// ---- Interfaces/I_ManualTarget.TcIO
// Core §7.6.1 — a module that can be commanded by hand, reached by the SAME
// deterministic walk that already carries configuration writes (I_ConfigSource).
//
// This exists because the walk was missing and every Unit hand-wrote its own
// routing instead:
//
//     IF TargetPath = PressRam.Name THEN _M_RouteManual := PressRam.ManualCommand(...)
//     ELSIF TargetPath = Door.Name  THEN ...
//
// That is a call a project has to remember for correctness, which §1.1 O1 names
// as a framework defect rather than a project style. It failed exactly the way
// O1 predicts: the press registered eight children and routed three, so the
// feed axis, the two-hand control, the power group, the part sensor and the air
// monitor all published manual commands that the HMI rendered as buttons and
// the Unit refused, with no diagnostic anybody could act on. Nothing was wrong
// with those modules; the routing chain simply had no branch for them.
//
// Configuration never had this problem because it was built as a capability
// walk from the start: a module answers for its own Scope and the composite
// recurses. Manual commands now use the identical shape, so a registered child
// is commandable BECAUSE it is registered, and a new module type costs no
// routing code anywhere.
INTERFACE I_ManualTarget EXTENDS __System.IQueryInterface

// Apply one one-shot manual command to the module named by Scope. TRUE only
// from the module that owns the path AND accepted the value, so the walk
// continues past every module that is not the target. The owning module still
// validates the command against its own published catalogue (§5.6) — this
// carries the request, it does not privilege it.
METHOD M_ApplyManual : BOOL
VAR_INPUT
    Scope : STRING(255);
    Value : DINT;
END_VAR
END_METHOD

// §7.6.1a — apply one HELD manual request (hold-to-run) to the module named by
// Scope, carrying the enabling-device status the root derived from its §9
// safety facet.
//
// Enable travels WITH the request rather than being read by the module, because
// the fact belongs to the safety system and the root is where it is mirrored.
// A module that does not implement held commands inherits FB_ModuleBase's
// refusal, so an unsupported hold is a defined FALSE and never a silent no-op.
METHOD M_ApplyHeld : BOOL
VAR_INPUT
    Scope  : STRING(255);
    Value  : DINT;
    Enable : ST_ManualEnableStatus;
END_VAR
END_METHOD

END_INTERFACE

// ---- Interfaces/I_Module.TcIO
// Core §3.2 — everything a parent needs to discover, monitor, and roll up a child.
// Reconciliation vs. Core §3.2 text: no ErrorID property here (it would collide with
// the PLCopen ErrorID output every module exposes, Core §6.1); callers read
// GetFaultSummary().ReasonCode. GetFaultSummary returns ST_Diagnostic (Core §8.8),
// Recipe changeover is a prepare/commit/abort transaction (Core §3.8).
INTERFACE I_Module EXTENDS __System.IQueryInterface

METHOD Cyclic : BOOL
END_METHOD

// recursive first-out walk (Core §8.2, §6.9)
METHOD GetFaultSummary : ST_Diagnostic
END_METHOD

// Load/validate into staging only; active ParCfg remains unchanged.
METHOD PrepareRecipe : BOOL
VAR_INPUT
    Model : ST_ModelId;
END_VAR
END_METHOD

// Infallible bounded publication after a successful PrepareRecipe.
METHOD CommitRecipe
END_METHOD

METHOD AbortRecipe
END_METHOD

// Core §6.1/§8.3(b) — release a command the owner can no longer complete, so the
// inherited Execute-drop reset can clear a latched terminal state. A parent needs
// this generically: when a mode chain freezes on a fault it stops polling the
// children it commanded, and a child whose Execute stays asserted can never be
// re-issued (no rising edge) nor reset (the drop reset needs Execute low).
METHOD M_ReleaseCommand : BOOL
END_METHOD

PROPERTY FaultActive : BOOL
GET
END_GET
END_PROPERTY

// Core §6.1 — TRUE while the module is BUSY but deliberately not progressing
// because a declared condition is unsatisfied (ISA-88 HELD). It is NOT a fault:
// outputs are withdrawn, the reason is published at LOW severity, and progress
// resumes by itself when the condition returns. The parent reads this to explain
// the wait instead of reporting a generic stall (§6.9).
PROPERTY HoldActive : BOOL
GET
END_GET
END_PROPERTY

PROPERTY ModuleType : E_ModuleType
GET
END_GET
END_PROPERTY

PROPERTY Name : STRING(80)
GET
END_GET
END_PROPERTY

PROPERTY State : E_ExecState
GET
END_GET
END_PROPERTY

END_INTERFACE

// ---- Interfaces/I_Sequence.TcIO
// Core §6.8 — the sliver of a step chain its OWNER needs.
// A chain receives the host bridge at Setup (I_SequenceHost); this is the
// reverse direction, so FB_UnitBase can drive scan-scoped housekeeping for
// every attached chain without the project wiring a single call.
INTERFACE I_Sequence

// §6.10 one-scan reset of the shared transition result.
METHOD M_BeginScan
END_METHOD

// §6.8 the chain starts over at its first step, application state included
// (OnChainReset). Driven by the owning Unit at the transitions after which a
// chain can never resume: first scan, mode change, abort.
METHOD M_Restart
END_METHOD

// §6.9 the owning Unit left ERROR: re-arm the step that raised it so the
// chain re-evaluates the command state instead of resuming mid-handshake.
METHOD M_ResumeAfterError
END_METHOD

END_INTERFACE

// ---- Interfaces/I_SequenceHost.TcIO
// Core §6.7/§6.8 — the bridge from a separately-compiled sequence POU (SFC/ST/LD)
// to its owning module's protected framework services: step record, condition
// waits, run-style gate, part lifecycle, decisions, and completion/fault.
// FB_UnitBase implements it once; a sequence receives it at Setup. It carries
// framework plumbing ONLY — application decisions stay in the sequence's steps.
INTERFACE I_SequenceHost

// §6.11 publish a decision request
METHOD M_SequenceAskDecision
VAR_INPUT
    Req : ST_DecisionRequest;
END_VAR
END_METHOD

// §6.9(b) named plain-condition wait
METHOD M_SequenceAwait : BOOL
VAR_INPUT
    Idx : INT;
    Label : STRING(120);
    Ok : BOOL;
END_VAR
END_METHOD

// §6.11 withdraw an open request
METHOD M_SequenceClearDecision
END_METHOD

// §6.1 one-shot sequence completion (finite chains)
METHOD M_SequenceComplete
END_METHOD

// §8.11.2 carrier-less fallback counter
METHOD M_SequenceCountGood
END_METHOD

// §8.11.1 cycle-complete marker; FALSE = stop granted (chain must not loop)
METHOD M_SequenceEndOfCycle : BOOL
END_METHOD

// §6.9 first-out fault from a step
METHOD M_SequenceFault
VAR_INPUT
    Reason : E_Reason;
    DescriptionKey : STRING(255);
END_VAR
END_METHOD

// §3.16.3 EVENT_PART_PROCESSED (write-result-first; counts by verdict §8.11.2)
METHOD M_SequencePartProcessed : BOOL
VAR_INPUT
    Verdict : E_Verdict;
    Reason : E_Reason;
END_VAR
END_METHOD

// §3.16.3 EVENT_PART_RECEIVED
METHOD M_SequencePartReceived : BOOL
END_METHOD

// §3.16.1 measured value
METHOD M_SequencePartRecord : BOOL
VAR_INPUT
    RecordName : STRING(64);
    Value : LREAL;
    Minimum : LREAL;
    Maximum : LREAL;
    Target : LREAL;
    EngUnit : STRING(16);
END_VAR
END_METHOD

// §3.16.3 EVENT_PART_PROCESSING_STARTED
METHOD M_SequencePartStarted
END_METHOD

// §6.8 a chain announces itself at M_Attach so the owning Unit can run
// scan-scoped housekeeping for it. Idempotent: Setup may run more than once.
METHOD M_SequenceRegister : BOOL
VAR_INPUT
    Seq : I_Sequence;
END_VAR
END_METHOD

// §6.9 raise a first-out from a step, with the module path the §3.13 flow
// chart links to. Unlike M_SequenceFault this carries severity/category and a
// link, so a step can adopt a child's fault verbatim or declare its own message.
METHOD M_SequenceRaise : BOOL
VAR_INPUT
    Diag     : ST_Diagnostic;
    LinkPath : STRING(255);
END_VAR
END_METHOD

// §6.9(e) publish a message that informs and does NOT stop the chain: an
// AUTO_RESET come+gone event (§8.3(c)) plus the §3.13 flow-chart row mark.
METHOD M_SequenceWarn : BOOL
VAR_INPUT
    Diag : ST_Diagnostic;
END_VAR
END_METHOD

// §6.5 step record (feeds the §6.9 walk and the §8.11.4 profiler)
METHOD M_SequenceSetStep
VAR_INPUT
    StepNo : INT;
    StepName : STRING(120);
    Awaits : I_Module;
    AwaitingLabel : STRING(120);
    TimeClass : E_TimeClass;
    ExpectedTime : TIME;
    Branch : INT;                  // §6.12 concurrent leg, 0 = main line
END_VAR
END_METHOD

// §3.4.2 run-style pacing gate
METHOD M_SequenceStepGate : BOOL
VAR_INPUT
    Steppable : BOOL;
END_VAR
END_METHOD

// §3.4/§8.11 — accept a pending Stop BETWEEN cycles: abandon the open cycle
// profile (no §8.11.1 cycle is counted for a wait-only fragment) and complete.
METHOD M_SequenceStopNow
END_METHOD

// §3.4 — TRUE while a Stop is requested and the sequence still runs. A chain
// polls this at its between-cycles wait so a stop need not ride out a phantom cycle.
METHOD M_SequenceStopPending : BOOL
END_METHOD

// §6.11 consume the answer once (0 = none yet)
METHOD M_SequenceTakeDecision : INT
END_METHOD

END_INTERFACE

// ---- Interfaces/I_RecipeStore.TcIO
// Core §3.8a - a recipe provider whose records can be edited. Optional: a provider
// that implements it lets a root edit the recipe of ANY model it offers, not only
// the active one, and keeps an edit of the active model across a changeover.
// Found by __QUERYINTERFACE on the I_RecipeProvider a module was given.
INTERFACE I_RecipeStore

// Replace the record of exactly (ModelCode, RecipeKey) with Size bytes at pData.
// FALSE when that record does not exist or its size or SchemaVersion differs:
// a fallback record is never edited in a specific model's name.
METHOD Save : BOOL
VAR_INPUT
    ModelCode : STRING;
    RecipeKey : STRING;
    pData     : PVOID;
    Size      : UDINT;
END_VAR
END_METHOD

END_INTERFACE

// ---- Interfaces/I_RecipeProvider.TcIO
// Core §3.8 — pluggable recipe/type-data source. Implementations MUST validate
// completeness and SchemaVersion before filling ParCfg (migrate-or-fault; never partial).
// Queryable (like I_Module) so a root can ask a provider for I_RecipeStore (§3.8a).
INTERFACE I_RecipeProvider EXTENDS __System.IQueryInterface

// fills the caller's ParCfg; FALSE => caller faults with RECIPE_INVALID (Core §3.8)
METHOD Load : BOOL
VAR_INPUT
    ModelCode : STRING;
    RecipeKey : STRING;
    pParCfg : PVOID;
    Size    : UDINT;
END_VAR
END_METHOD

PROPERTY Ready : BOOL
GET
END_GET
END_PROPERTY

PROPERTY Source : E_RecipeSource
GET
END_GET
END_PROPERTY

END_INTERFACE

// ---- Connectivity/FB_LocalRecipeProvider.TcPOU
// Core §3.8 local provider. Validation is generic BECAUSE SchemaVersion is the
// first UINT of every ParCfg/record (§3.8): stored first-UINT must equal the
// target's initialized first-UINT, else Load = FALSE and the caller faults
// RECIPE_INVALID. Never a partial apply. Types stage through PrepareRecipe.
FUNCTION_BLOCK FB_LocalRecipeProvider IMPLEMENTS I_RecipeProvider, I_RecipeStore, I_RecipeCatalog
VAR PERSISTENT
    {attribute 'OPC.UA.DA' := '0'}
    _catalog : ST_LocalRecipeCatalog;
END_VAR
VAR
    _catalogInitialized : BOOL;
    _catalogRestoreVersion : UINT;
    _n    : INT;
    _models : ARRAY[1..PL_Fraktal.MAX_RECIPES] OF STRING(80);
    _keys   : ARRAY[1..PL_Fraktal.MAX_RECIPES] OF STRING(80);
    {attribute 'OPC.UA.DA' := '0'}
    _ptr  : ARRAY[1..PL_Fraktal.MAX_RECIPES] OF PVOID;
    _size : ARRAY[1..PL_Fraktal.MAX_RECIPES] OF UDINT;
END_VAR

// no cyclic body

METHOD Load : BOOL
VAR_INPUT
    ModelCode : STRING;
    RecipeKey : STRING;
    pParCfg : PVOID;
    Size    : UDINT;
END_VAR
VAR
    i, hit, fallback : INT;
    puT, puS : POINTER TO UINT;
END_VAR
_M_InitCatalog();
Load := FALSE;
IF (pParCfg = 0) OR (Size < SIZEOF(puT^)) THEN RETURN; END_IF
FOR i := 1 TO _catalog.Count DO
    IF (_catalog.Records[i].ModelCode = ModelCode)
    AND (_catalog.Records[i].RecipeKey = RecipeKey) THEN
        IF _catalog.Records[i].DataSize <> Size THEN RETURN; END_IF
        puT := pParCfg;
        puS := ADR(_catalog.Records[i].Data);
        IF puT^ <> puS^ THEN RETURN; END_IF
        MEMCPY(destAddr := pParCfg,
            srcAddr := ADR(_catalog.Records[i].Data), n := Size);
        Load := TRUE;
        RETURN;
    END_IF
END_FOR
hit := 0;
fallback := 0;
FOR i := 1 TO _n DO
    IF (_keys[i] = RecipeKey) AND (_models[i] = ModelCode) THEN
        hit := i;
        EXIT;
    ELSIF (_keys[i] = RecipeKey) AND (_models[i] = '') THEN
        fallback := i;
    END_IF
END_FOR
IF hit = 0 THEN
    hit := fallback;
END_IF
// Two statements, not one condition: IEC 61131-3 does not mandate short-circuit
// evaluation and TwinCAT's compile option for it is off by default, so a single
// `(hit = 0) OR (_size[hit] <> Size)` still reads _size[0] on the ordinary
// not-found path - out of bounds for ARRAY[1..MAX_RECIPES] (§3.8).
IF (hit = 0) OR (pParCfg = 0) THEN
    RETURN;                                       // unknown recipe -> caller faults (§3.8)
END_IF
IF _size[hit] <> Size THEN
    RETURN;                                       // size mismatch -> caller faults (§3.8)
END_IF
puT := pParCfg;
puS := _ptr[hit];
IF puT^ <> puS^ THEN
    RETURN;                                       // SchemaVersion mismatch: migrate-or-fault (§3.8)
END_IF
MEMCPY(destAddr := pParCfg, srcAddr := _ptr[hit], n := Size);
Load := TRUE;
END_METHOD

// I_RecipeStore - write an edited record back into the registered storage of
// exactly (ModelCode, RecipeKey). The fallback record is never edited in a
// specific model's name, and a size or SchemaVersion mismatch changes nothing.
METHOD Save : BOOL
VAR_INPUT
    ModelCode : STRING;
    RecipeKey : STRING;
    pData     : PVOID;
    Size      : UDINT;
END_VAR
VAR
    i, hit : INT;
    puT, puS : POINTER TO UINT;
END_VAR
_M_InitCatalog();
Save := FALSE;
IF (pData = 0) OR (Size < SIZEOF(puT^)) THEN RETURN; END_IF
FOR i := 1 TO _catalog.Count DO
    IF (_catalog.Records[i].ModelCode = ModelCode)
    AND (_catalog.Records[i].RecipeKey = RecipeKey) THEN
        IF _catalog.Records[i].DataSize <> Size THEN RETURN; END_IF
        puT := pData;
        puS := ADR(_catalog.Records[i].Data);
        IF puT^ <> puS^ THEN RETURN; END_IF
        MEMCPY(destAddr := ADR(_catalog.Records[i].Data),
            srcAddr := pData, n := Size);
        Save := TRUE;
        RETURN;
    END_IF
END_FOR
hit := 0;
FOR i := 1 TO _n DO
    IF (_keys[i] = RecipeKey) AND (_models[i] = ModelCode) THEN
        hit := i;
        EXIT;
    END_IF
END_FOR
IF (hit = 0) OR (pData = 0) THEN
    RETURN;
END_IF
IF _size[hit] <> Size THEN
    RETURN;
END_IF
puT := _ptr[hit];
puS := pData;
IF puT^ <> puS^ THEN
    RETURN;                                       // SchemaVersion differs: nothing written
END_IF
MEMCPY(destAddr := _ptr[hit], srcAddr := pData, n := Size);
Save := TRUE;
END_METHOD

// application wiring: one record per (ModelCode, RecipeKey); empty ModelCode is fallback.
METHOD Register : BOOL
VAR_INPUT
    ModelCode : STRING(80);
    RecipeKey : STRING(80);
    pData  : PVOID;
    Size   : UDINT;
END_VAR
VAR
    i : INT;
END_VAR
_M_InitCatalog();
IF (_n + _catalog.Count >= PL_Fraktal.MAX_RECIPES) OR (pData = 0) OR (RecipeKey = '') OR (Size < SIZEOF(UINT)) THEN
    Register := FALSE;
    RETURN;
END_IF
FOR i := 1 TO _n DO
    IF (_models[i] = ModelCode) AND (_keys[i] = RecipeKey) THEN
        Register := FALSE;
        RETURN;
    END_IF
END_FOR
FOR i := 1 TO _catalog.Count DO
    IF (_catalog.Records[i].ModelCode = ModelCode)
    AND (_catalog.Records[i].RecipeKey = RecipeKey) THEN
        Register := FALSE;
        RETURN;
    END_IF
END_FOR
_n := _n + 1;
_models[_n] := ModelCode;
_keys[_n]   := RecipeKey;
_ptr[_n]  := pData;
_size[_n] := Size;
Register := TRUE;
END_METHOD

PROPERTY Ready : BOOL
GET
Ready := (_n > 0);
END_GET
END_PROPERTY

PROPERTY Source : E_RecipeSource
GET
Source := E_RecipeSource.LOCAL;
END_GET
END_PROPERTY

METHOD PRIVATE _M_InitCatalog
VAR
    i, j : INT;
    schema : UINT;
    pSchema : POINTER TO UINT;
    valid : BOOL;
END_VAR
IF _catalogInitialized THEN RETURN; END_IF
_catalogInitialized := TRUE;
IF (_catalog.SchemaVersion = 1) AND (_catalog.Count >= 0)
AND (_catalog.Count <= PL_Fraktal.MAX_RECIPES) THEN
    valid := TRUE;
    FOR i := 1 TO _catalog.Count DO
        IF (_catalog.Records[i].SchemaVersion <> 1)
        OR (_catalog.Records[i].ModelCode = '') OR (_catalog.Records[i].RecipeKey = '')
        OR (_catalog.Records[i].DataSize < SIZEOF(schema))
        OR (_catalog.Records[i].DataSize > PL_Fraktal.MAX_MODEL_DATA_BYTES) THEN
            valid := FALSE;
        END_IF
        pSchema := ADR(_catalog.Records[i].Data);
        IF pSchema^ = 0 THEN valid := FALSE; END_IF
        FOR j := 1 TO i - 1 DO
            IF _catalog.Records[i].ModelCode = _catalog.Records[j].ModelCode THEN
                valid := FALSE;
            END_IF
        END_FOR
    END_FOR
    IF valid THEN RETURN; END_IF
END_IF
IF _catalog.SchemaVersion <> 0 THEN
    _catalogRestoreVersion := _catalog.SchemaVersion;
END_IF
_catalog.Count := 0;
_catalog.SchemaVersion := 1;
END_METHOD

METHOD M_ModelCount : INT
VAR_INPUT
    RecipeKey : STRING(80);
END_VAR
VAR
    i : INT;
END_VAR
_M_InitCatalog();
M_ModelCount := 0;
FOR i := 1 TO _n DO
    IF (_keys[i] = RecipeKey) AND (_models[i] <> '') THEN
        M_ModelCount := M_ModelCount + 1;
    END_IF
END_FOR
FOR i := 1 TO _catalog.Count DO
    IF _catalog.Records[i].RecipeKey = RecipeKey THEN
        M_ModelCount := M_ModelCount + 1;
    END_IF
END_FOR
END_METHOD

METHOD M_ModelCapacity : INT
VAR_INPUT
    RecipeKey : STRING(80);
END_VAR
VAR
    i : INT;
END_VAR
_M_InitCatalog();
M_ModelCapacity := M_ModelCount(RecipeKey := RecipeKey)
    + PL_Fraktal.MAX_RECIPES - _n - _catalog.Count;
// Released seed registration accepts 80 bytes; the root identity accepts 64.
// Preserve that API while refusing a catalog projection that would truncate it.
FOR i := 1 TO _n DO
    IF (_keys[i] = RecipeKey) AND (LEN(_models[i]) > 64) THEN
        M_ModelCapacity := 0; RETURN;
    END_IF
END_FOR
END_METHOD

METHOD M_ModelAt : BOOL
VAR_INPUT
    RecipeKey : STRING(80);
    Index : INT;
END_VAR
VAR_IN_OUT
    Id : ST_ModelId;
END_VAR
VAR
    i, ordinal : INT;
END_VAR
_M_InitCatalog();
M_ModelAt := FALSE;
IF Index < 1 THEN RETURN; END_IF
ordinal := 0;
FOR i := 1 TO _n DO
    IF (_keys[i] = RecipeKey) AND (_models[i] <> '') THEN
        ordinal := ordinal + 1;
        IF ordinal = Index THEN
            IF LEN(_models[i]) > 64 THEN RETURN; END_IF
            Id.ModelCode := _models[i];
            M_ModelAt := TRUE;
            RETURN;
        END_IF
    END_IF
END_FOR
FOR i := 1 TO _catalog.Count DO
    IF _catalog.Records[i].RecipeKey = RecipeKey THEN
        ordinal := ordinal + 1;
        IF ordinal = Index THEN
            Id.ModelCode := _catalog.Records[i].ModelCode;
            M_ModelAt := TRUE;
            RETURN;
        END_IF
    END_IF
END_FOR
END_METHOD

METHOD M_CreateModel : BOOL
VAR_INPUT
    ModelCode : STRING(64);
    RecipeKey : STRING(80);
    pData : PVOID;
    Size : UDINT;
END_VAR
VAR
    i, slot : INT;
    pSchema : POINTER TO UINT;
END_VAR
_M_InitCatalog();
M_CreateModel := FALSE;
IF (ModelCode = '') OR (RecipeKey = '') OR (pData = 0)
OR (Size < SIZEOF(pSchema^)) OR (Size > PL_Fraktal.MAX_MODEL_DATA_BYTES)
OR (_n + _catalog.Count >= PL_Fraktal.MAX_RECIPES) THEN RETURN; END_IF
pSchema := pData;
IF pSchema^ = 0 THEN RETURN; END_IF
FOR i := 1 TO _n DO
    IF _models[i] = ModelCode THEN RETURN; END_IF
END_FOR
FOR i := 1 TO _catalog.Count DO
    IF _catalog.Records[i].ModelCode = ModelCode THEN RETURN; END_IF
END_FOR
slot := _catalog.Count + 1;
_catalog.Records[slot].SchemaVersion := 1;
_catalog.Records[slot].ModelCode := ModelCode;
_catalog.Records[slot].RecipeKey := RecipeKey;
_catalog.Records[slot].DataSize := Size;
MEMCPY(destAddr := ADR(_catalog.Records[slot].Data), srcAddr := pData, n := Size);
_catalog.Count := slot; // publication LAST; every existing address stays stable
M_CreateModel := TRUE;
END_METHOD

METHOD M_TakeCatalogRestoreLoss : BOOL
VAR_OUTPUT
    Found : UINT;
END_VAR
_M_InitCatalog();
Found := _catalogRestoreVersion;
M_TakeCatalogRestoreLoss := Found <> 0;
_catalogRestoreVersion := 0;
END_METHOD

END_FUNCTION_BLOCK

// ---- Connectivity/FB_LocalAccessProvider.TcPOU
// Core §7.7(c) — DEFAULT local provider: a durable user table. Remote/central
// auth (server, LDAP via gateway) substitutes behind I_AccessProvider later.
//
// §14 - a PIN is never stored: each user keeps a random-per-registration salt and
// an iterated SHA-256 of salt and PIN, and the table is hidden from the ADS symbol
// table and OPC UA. Hiding is the control that matters for a short PIN - four
// digits fall to an offline search whatever the hash - so the hash's job is that a
// dump, backup or retained file does not hand the PINs out as text.
//
// TwinCAT restores PERSISTENT data by symbol and a hidden variable has none, so a
// hidden table cannot be PERSISTENT (IMPLEMENTATION_NOTES §154). The table is kept
// instead as one CRC-protected image document on an I_PersistMedium (§163): by
// default a file medium in the runtime's TwinCAT Boot directory, or the project's
// own medium (M_UseMedium) - which must be confidential, so a retentive-memory
// pool, readable over ADS, is refused. The medium keeps two copies, never
// overwrites the newest, and reports a document it confirmed and then lost. The
// owning root's FB_AccessManager drives restore and save through I_AccessStore
// every scan: a project calls nothing to make its users durable.
{attribute 'reflection'}
FUNCTION_BLOCK FB_LocalAccessProvider IMPLEMENTS I_AccessProvider, I_AccessStore
VAR_OUTPUT
    Restored     : BOOL;    // the retained table has been read (or there was none)
    Durable      : BOOL;    // every registration so far is in a written image
    StorageError : UDINT;   // last medium error (0 = none)
END_VAR
VAR
    {attribute 'hide'}
    {attribute 'OPC.UA.DA' := '0'}
    _users : ARRAY[1..PL_Fraktal.MAX_USERS] OF ST_UserRecord;
    {attribute 'hide'}
    {attribute 'OPC.UA.DA' := '0'}
    _n     : INT;
    {attribute 'hide'}
    _saltSeq : UDINT;
    // Transfer buffer: the image read, then each image written. It carries salts
    // and hashes, so it is hidden like the table; the medium only borrows it.
    {attribute 'hide'}
    {attribute 'OPC.UA.DA' := '0'}
    _image : ST_AccessImageV1;
    // '<project>.<path>.<instance>': hashed into the default key, so two providers -
    // or two PLC projects on one runtime - never share a document.
    {attribute 'instance-path'}
    {attribute 'noinit'}
    _instancePath : STRING(255);
    _key         : STRING(80);
    _keyChosen   : BOOL;            // the key is decided (possibly '' = volatile)
    {attribute 'OPC.UA.DA' := '0'}
    _medium      : I_PersistMedium; // injected, or _ownMedium
    {attribute 'OPC.UA.DA' := '0'}
    _ownMedium   : FB_FilePersistMedium;
    _ticket      : UDINT;
    _result      : ST_PersistResult;
    _phase       : INT;
    _generation  : UDINT;           // generation of the newest image written or read
    _restoreLost : BOOL;
    _dirty       : BOOL;            // the table changed since the last written image
    _changeSeq   : UDINT;
    _writeSeq    : UDINT;           // _changeSeq captured into the image being written
    _saveFailed  : BOOL;
    _readFailed  : BOOL;            // the medium could not answer the restore read
    _retry       : TON;
END_VAR
VAR CONSTANT
    IMAGE_MAGIC    : DWORD := DWORD#16#414B5246;   // 'FRKA', little endian
    RETRY_INTERVAL : TIME := T#10S;
END_VAR

// no cyclic body: the owning root's FB_AccessManager calls M_Service

// Keep the table on the project's medium instead of the Boot directory - the
// same instance the project gives its roots, so one line switches every
// retained document. Refused: no medium, a medium that is not confidential
// (a credential never becomes symbol-readable, §14), or a restore already begun.
METHOD M_UseMedium : BOOL
VAR_INPUT
    Medium : I_PersistMedium;
END_VAR
M_UseMedium := FALSE;
IF (_phase <> 0) OR (Medium = 0) THEN
    RETURN;
END_IF
IF NOT Medium.M_Confidential() THEN
    RETURN;
END_IF
_medium := Medium;
M_UseMedium := TRUE;
END_METHOD

// The table's document key on the medium (a file medium stores '<key>.a' and
// '<key>.b'). Without a call it is 'FraktalAccess_' and the CRC of this
// instance's path, so two providers - or two PLC projects on one runtime - never
// share a document. '' keeps the table volatile (a fixture, or a station whose
// users come from elsewhere). Letters, digits, '_', '.' and '-'. Refused once
// the restore has started: retargeting a live store would split one table.
METHOD M_UseKey : BOOL
VAR_INPUT
    Key : STRING(80);
END_VAR
M_UseKey := FALSE;
IF _phase <> 0 THEN
    RETURN;
END_IF
IF (Key <> '') AND NOT F_ValidPersistKey(Key := Key) THEN
    RETURN;
END_IF
_key := Key;
_keyChosen := TRUE;
M_UseKey := TRUE;
END_METHOD

// I_AccessStore - read the table's image once, then keep the written image
// current. A second root sharing this provider merely advances the same steps.
METHOD M_Service : BOOL
CASE _phase OF
    0:
        IF NOT _keyChosen THEN
            _key := _M_DefaultKey();
            _keyChosen := TRUE;
        END_IF
        IF _key = '' THEN
            Restored := TRUE;       // volatile by choice: nothing to restore or save
            Durable := FALSE;
            _phase := 90;
        ELSE
            IF _medium = 0 THEN
                _ownMedium.Setup(Folder := '', Where := Tc2_System.PATH_BOOTPATH);
                _medium := _ownMedium;
            END_IF
            _phase := 10;
        END_IF
    10:     // ask for the image
        MEMSET(destAddr := ADR(_image), fillByte := 0, n := SIZEOF(_image));
        _ticket := _medium.M_StartRead(Key := _key, pData := ADR(_image),
            Size := SIZEOF(_image));
        IF _ticket <> 0 THEN
            _phase := 11;
        END_IF
    11:
        IF _medium.M_Poll(Ticket := _ticket, Result := _result) THEN
            IF _result.Ok THEN
                _readFailed := FALSE;
                _M_FinishRestore();
                _phase := 30;
            ELSE
                // Not "no table": the medium could not answer. Asked again; until
                // then nothing is merged, written or claimed lost.
                _readFailed := TRUE;
                StorageError := _result.ErrorId;
                _retry(IN := FALSE, PT := RETRY_INTERVAL);
                _phase := 12;
            END_IF
        END_IF
    12:
        _retry(IN := TRUE, PT := RETRY_INTERVAL);
        IF _retry.Q THEN
            _retry(IN := FALSE, PT := RETRY_INTERVAL);
            _phase := 10;
        END_IF
    30:     // idle: rewrite the table whenever it changed
        _retry(IN := _saveFailed, PT := RETRY_INTERVAL);
        IF _dirty AND (NOT _saveFailed OR _retry.Q) THEN
            _retry(IN := FALSE, PT := RETRY_INTERVAL);
            _M_BuildImage();
            _phase := 40;
        END_IF
    40:
        _ticket := _medium.M_StartWrite(Key := _key, pData := ADR(_image),
            Size := SIZEOF(_image));
        IF _ticket <> 0 THEN
            _phase := 41;
        END_IF
    41:
        IF _medium.M_Poll(Ticket := _ticket, Result := _result) THEN
            _M_SaveDone(Ok := _result.Ok);
            _phase := 30;
        END_IF
    90:
        ;   // volatile: the table lives for this run only
ELSE
    _phase := 30;   // unknown step: idle again; a pending change is rewritten
END_CASE
M_Service := Restored;
END_METHOD

// Decide what the medium answered. A restore LOST something when the medium
// reports a document it confirmed and lost, when the image it returned does not
// validate, or when the image's users no longer fit. Nothing there and nothing
// confirmed is a first start. (A medium that could not answer is asked again.)
METHOD PRIVATE _M_FinishRestore
StorageError := _result.ErrorId;
_restoreLost := _result.Lost;
IF _result.Found THEN
    IF (_result.Length = SIZEOF(_image)) AND _M_ValidImage(Image := _image) THEN
        _generation := _image.Generation;
        IF NOT _M_Merge() THEN
            _restoreLost := TRUE;
        END_IF
    ELSE
        _restoreLost := TRUE;       // a document this build cannot read as a table
    END_IF
END_IF
MEMSET(destAddr := ADR(_image), fillByte := 0, n := SIZEOF(_image));
IF _restoreLost THEN
    // Write what survived as the new baseline: the loss is announced once, not at
    // every restart.
    _M_Changed();
END_IF
Restored := TRUE;
Durable := NOT _dirty;
END_METHOD

// A change made while the image was being written is newer than that image, so
// the table stays dirty and is written again.
METHOD PRIVATE _M_SaveDone
VAR_INPUT
    Ok : BOOL;
END_VAR
IF Ok THEN
    _generation := _image.Generation;
    _saveFailed := FALSE;
    StorageError := 0;
    IF _changeSeq = _writeSeq THEN
        _dirty := FALSE;
    END_IF
ELSE
    _saveFailed := TRUE;    // retried; the medium never overwrites the newest copy
    StorageError := _result.ErrorId;
END_IF
MEMSET(destAddr := ADR(_image), fillByte := 0, n := SIZEOF(_image));
Durable := NOT _dirty AND NOT _saveFailed;
END_METHOD

// 'FraktalAccess_' + the CRC-32 of this instance's path, in hexadecimal.
METHOD PRIVATE _M_DefaultKey : STRING(80)
VAR
    pathLength : UDINT;
END_VAR
pathLength := INT_TO_UDINT(LEN(_instancePath));
_M_DefaultKey := CONCAT('FraktalAccess_', Tc2_Utilities.DWORD_TO_HEXSTR(
    in := F_Crc32(pData := ADR(_instancePath), Size := pathLength),
    iPrecision := 8, bLoCase := FALSE));
END_METHOD

METHOD Authenticate : E_AccessLevel
VAR_INPUT
    User : STRING(32);
    Secret : STRING(32);
END_VAR
VAR
    i : INT;
    hit : INT;
    noSalt : ARRAY[0..15] OF BYTE;
    candidate : ARRAY[0..31] OF BYTE;
    diff : BYTE;
    k : INT;
END_VAR
Authenticate := E_AccessLevel.NONE;
hit := 0;
FOR i := 1 TO _n DO
    IF _users[i].User = User THEN
        hit := i;
    END_IF
END_FOR
IF hit = 0 THEN
    // An unknown user costs the same hash, so timing does not tell names apart.
    _M_Hash(Salt := noSalt, Pin := Secret, Digest := candidate);
    RETURN;
END_IF
_M_Hash(Salt := _users[hit].Salt, Pin := Secret, Digest := candidate);
diff := 0;
FOR k := 0 TO 31 DO
    diff := diff OR (candidate[k] XOR _users[hit].PinHash[k]);
END_FOR
IF diff = 0 THEN
    Authenticate := _users[hit].Level;
END_IF
END_METHOD

// commissioning-time user entry (itself an ACCESS_POLICY-gated edit via the HMI).
// Idempotent by User: re-registering replaces PIN/level, and the retained table
// keeps the user, so a composition root may register its defaults every boot
// without duplicates. Every registration draws a new salt. A registration made
// before the restore completes is kept and wins over the retained record.
// Refused: an empty name, a level outside NONE..ADMIN, or a full table.
METHOD Register : BOOL
VAR_INPUT
    User : STRING(32);
    Pin : STRING(32);
    Level : E_AccessLevel;
END_VAR
VAR
    i : INT;
    slot : INT;
END_VAR
Register := FALSE;
IF (User = '') OR (TO_DINT(Level) < TO_DINT(E_AccessLevel.NONE))
OR (TO_DINT(Level) > TO_DINT(E_AccessLevel.ADMIN)) THEN
    RETURN;     // an image holding such a record would be refused at restore
END_IF
slot := 0;
FOR i := 1 TO _n DO
    IF _users[i].User = User THEN
        slot := i;
    END_IF
END_FOR
IF slot = 0 THEN
    IF _n >= PL_Fraktal.MAX_USERS THEN
        RETURN;
    END_IF
    _n := _n + 1;
    slot := _n;
    _users[slot].User := User;
END_IF
_M_NewSalt(User := User, Salt := _users[slot].Salt);
_M_Hash(Salt := _users[slot].Salt, Pin := Pin, Digest := _users[slot].PinHash);
_users[slot].Level := Level;
_M_Changed();
Register := TRUE;
END_METHOD

METHOD M_RestoreLost : BOOL
M_RestoreLost := _restoreLost;
END_METHOD

METHOD M_SaveFailed : BOOL
M_SaveFailed := _saveFailed OR _readFailed;
END_METHOD

// Add every retained user not registered in this run. A registration made before
// the restore finished is newer, so it stands. FALSE = a user did not fit.
METHOD PRIVATE _M_Merge : BOOL
VAR
    i : INT;
    k : INT;
    found : BOOL;
END_VAR
_M_Merge := TRUE;
FOR i := 1 TO _image.Count DO
    found := FALSE;
    FOR k := 1 TO _n DO
        IF _users[k].User = _image.Users[i].User THEN
            found := TRUE;
        END_IF
    END_FOR
    IF NOT found THEN
        IF _n < PL_Fraktal.MAX_USERS THEN
            _n := _n + 1;
            _users[_n] := _image.Users[i];
        ELSE
            _M_Merge := FALSE;
        END_IF
    END_IF
END_FOR
END_METHOD

// Whole-image validation: format, checksum, then every record. One bad record
// rejects the image - a table is restored completely or not at all.
METHOD PRIVATE _M_ValidImage : BOOL
VAR_IN_OUT
    Image : ST_AccessImageV1;
END_VAR
VAR
    i : INT;
    k : INT;
END_VAR
_M_ValidImage := FALSE;
IF (Image.SchemaVersion <> 1) OR (Image.ByteCount <> SIZEOF(Image))
OR (Image.Magic <> IMAGE_MAGIC) OR (Image.Reserved <> 0)
OR (Image.Count < 0) OR (Image.Count > PL_Fraktal.MAX_USERS) THEN
    RETURN;
END_IF
IF Image.Crc <> F_Crc32(pData := ADR(Image), Size := SIZEOF(Image) - SIZEOF(Image.Crc)) THEN
    RETURN;
END_IF
FOR i := 1 TO Image.Count DO
    IF (Image.Users[i].User = '')
    OR (TO_DINT(Image.Users[i].Level) < TO_DINT(E_AccessLevel.NONE))
    OR (TO_DINT(Image.Users[i].Level) > TO_DINT(E_AccessLevel.ADMIN)) THEN
        RETURN;
    END_IF
    FOR k := 1 TO i - 1 DO
        IF Image.Users[k].User = Image.Users[i].User THEN
            RETURN;
        END_IF
    END_FOR
END_FOR
_M_ValidImage := TRUE;
END_METHOD

METHOD PRIVATE _M_BuildImage
VAR
    i : INT;
END_VAR
MEMSET(destAddr := ADR(_image), fillByte := 0, n := SIZEOF(_image));
_image.SchemaVersion := 1;
_image.ByteCount := TO_UINT(SIZEOF(_image));
_image.Magic := IMAGE_MAGIC;
_image.Generation := _generation + 1;
_image.Count := _n;
FOR i := 1 TO _n DO
    _image.Users[i] := _users[i];
END_FOR
_image.Crc := F_Crc32(pData := ADR(_image), Size := SIZEOF(_image) - SIZEOF(_image.Crc));
_writeSeq := _changeSeq;
END_METHOD

METHOD PRIVATE _M_Changed
_dirty := TRUE;
_changeSeq := _changeSeq + 1;
Durable := FALSE;
END_METHOD

// A salt unique to this registration: the clock, a sequence and the user name,
// hashed. It need not be secret, only never repeated.
METHOD PRIVATE _M_NewSalt
VAR_INPUT
    User : STRING(32);
END_VAR
VAR_IN_OUT
    Salt : ARRAY[0..15] OF BYTE;
END_VAR
VAR
    seed : ARRAY[0..47] OF BYTE;
    now : ULINT;
    digest : ARRAY[0..31] OF BYTE;
END_VAR
now := Tc2_Utilities.F_GetSystemTime();
_saltSeq := _saltSeq + 1;
MEMCPY(destAddr := ADR(seed), srcAddr := ADR(now), n := SIZEOF(now));
MEMCPY(destAddr := ADR(seed) + 8, srcAddr := ADR(_saltSeq), n := SIZEOF(_saltSeq));
MEMCPY(destAddr := ADR(seed) + 12, srcAddr := ADR(User), n := INT_TO_UDINT(LEN(User)));
F_Sha256(pData := ADR(seed), Size := 12 + INT_TO_UDINT(LEN(User)), Digest := digest);
MEMCPY(destAddr := ADR(Salt), srcAddr := ADR(digest), n := 16);
END_METHOD

// SHA-256(Salt || Pin), then PL_Fraktal.PIN_HASH_ROUNDS more rounds of
// SHA-256(previous || Salt).
METHOD PRIVATE _M_Hash
VAR_INPUT
    Pin : STRING(32);
END_VAR
VAR_IN_OUT
    Salt   : ARRAY[0..15] OF BYTE;
    Digest : ARRAY[0..31] OF BYTE;
END_VAR
VAR
    buf : ARRAY[0..47] OF BYTE;
    round : UINT;
END_VAR
MEMCPY(destAddr := ADR(buf), srcAddr := ADR(Salt), n := 16);
MEMCPY(destAddr := ADR(buf) + 16, srcAddr := ADR(Pin), n := INT_TO_UDINT(LEN(Pin)));
F_Sha256(pData := ADR(buf), Size := 16 + INT_TO_UDINT(LEN(Pin)), Digest := Digest);
FOR round := 1 TO PL_Fraktal.PIN_HASH_ROUNDS DO
    MEMCPY(destAddr := ADR(buf), srcAddr := ADR(Digest), n := 32);
    MEMCPY(destAddr := ADR(buf) + 32, srcAddr := ADR(Salt), n := 16);
    F_Sha256(pData := ADR(buf), Size := 48, Digest := Digest);
END_FOR
MEMSET(destAddr := ADR(buf), fillByte := 0, n := SIZEOF(buf));
END_METHOD

END_FUNCTION_BLOCK

// ---- Platform/FB_FilePersistMedium.TcPOU
// Core §3.8b - the FILE medium (E_ConfigStore.FILE_JSON) on Tc2_System file
// services. Each key is two files in one folder, '<key>.a' and '<key>.b', and a
// write always replaces the slot NOT holding the newest valid copy, so a write
// cut short by a power loss leaves the previous document whole.
//
// Every file is an 80-byte text header line, then the document unchanged:
//   FRAKTAL-DOC 1 G=<generation> L=<length> K=<key CRC> C=<data CRC> H=<header CRC>
// in hexadecimal, so a set document stays readable in an editor. K binds a file
// to its key (a copy renamed to another key is refused), C checks the document
// and H the header. The highest valid generation wins on read.
//
// Both headers are read again before every write: the slot to replace and the
// next generation always come from what is on storage NOW, never from an earlier
// conclusion. A slot that cannot be READ (a file-service error other than "not
// found") is not a slot that is empty: a read then answers Ok = FALSE - the
// medium could not answer, nothing is claimed lost - and a write is refused
// without touching either file. Only content that reads but does not verify is
// treated as damaged.
//
// The generation each key was last CONFIRMED written at is kept PERSISTENT
// (it is not secret). A read that finds nothing valid where something was
// confirmed, or finds an older generation, reports Lost. TwinCAT stores the
// table at shutdown or on an explicit persistent write, so it can lag and never
// vouches for a write that did not happen; a stale marker can only miss a loss.
// The table is keyed by F_Crc32(folder + key), so retargeting the medium never
// claims a loss for files that were simply never written there. Keys beyond
// MAX_PERSIST_KEYS still work, without loss detection.
//
// Not symbol-readable: documents pass through the caller's buffer, so this
// medium may hold credentials (M_Confidential). On an IPC image with a write
// filter (UWF/EWF/FBWF), the folder must be excluded or every write reverts at
// the next boot. Files are created by the TwinCAT runtime's account; the
// folder's ACL decides who else may change them.
FUNCTION_BLOCK FB_FilePersistMedium EXTENDS FB_PersistMediumBase
VAR_OUTPUT
    StorageError : UDINT;   // last file-service error (0 = none)
END_VAR
VAR PERSISTENT
    {attribute 'OPC.UA.DA' := '0'}
    _confirmedKey : ARRAY[1..PL_Fraktal.MAX_PERSIST_KEYS] OF DWORD;
    {attribute 'OPC.UA.DA' := '0'}
    _confirmedGen : ARRAY[1..PL_Fraktal.MAX_PERSIST_KEYS] OF UDINT;
END_VAR
VAR
    _folder      : STRING(160);
    _where       : Tc2_System.E_OpenPath := Tc2_System.PATH_BOOTPATH;
    _foldersMade : BOOL;
    _mkPos       : INT;
    // The active request.
    _phase    : INT;
    _keyCrc   : DWORD;
    _slot     : INT;
    _hdrValid : ARRAY[1..2] OF BOOL;
    _hdrGen   : ARRAY[1..2] OF UDINT;
    _hdrLen   : ARRAY[1..2] OF UDINT;
    _hdrCrc   : ARRAY[1..2] OF DWORD;
    _invalidSeen : BOOL;    // a slot read but did not verify
    _ioFailed : BOOL;       // a slot could not be read at all
    _attempt  : INT;
    _ioOk     : BOOL;
    _handle   : UINT;
    _newGen   : UDINT;
    _header   : ARRAY[0..79] OF BYTE;   // read into / written from
    _expect   : ARRAY[0..79] OF BYTE;   // the header a read one must equal
    {attribute 'OPC.UA.DA' := '0'}
    _mkdir : Tc2_System.FB_CreateDir;
    {attribute 'OPC.UA.DA' := '0'}
    _open  : Tc2_System.FB_FileOpen;
    {attribute 'OPC.UA.DA' := '0'}
    _read  : Tc2_System.FB_FileRead;
    {attribute 'OPC.UA.DA' := '0'}
    _write : Tc2_System.FB_FileWrite;
    {attribute 'OPC.UA.DA' := '0'}
    _close : Tc2_System.FB_FileClose;
END_VAR
VAR CONSTANT
    HEADER_BYTES   : UDINT := 80;
    HEADER_TEXT    : STRING(80) := 'FRAKTAL-DOC 1 G=00000000 L=00000000 K=00000000 C=00000000 H=00000000';
    HEADER_CRC_SPAN : UDINT := 58;      // bytes before 'H='
    FILE_NOT_FOUND : UDINT := 16#70C;   // ADSERR_DEVICE_NOTFOUND
    CLOSE_DONE     : UDINT := 16#703;   // the handle is already released
    TOO_LARGE      : UDINT := 16#705;   // the document exceeds the caller's buffer
    IO_TIMEOUT     : TIME := T#3S;
END_VAR

// no cyclic body: every caller's M_Poll advances the medium

// Where the files live. Where = PATH_GENERIC takes an absolute Folder, for
// example 'C:\ProgramData\Fraktal\Station\'; PATH_BOOTPATH is relative to the
// TwinCAT Boot directory ('' = the directory itself). Missing folders are
// created on the first request. At most 160 characters; a trailing separator is
// added. Refused once a request was queued: one medium never splits a document
// over two folders.
METHOD Setup : BOOL
VAR_INPUT
    Folder : STRING(200);
    Where  : Tc2_System.E_OpenPath;
END_VAR
VAR
    n : INT;
    p : POINTER TO BYTE;
END_VAR
Setup := FALSE;
IF (_lastTicket > 0) OR (LEN(Folder) > 159) THEN
    RETURN;
END_IF
_folder := Folder;
n := LEN(_folder);
IF n > 0 THEN
    p := ADR(_folder);
    IF (p[n - 1] <> 92) AND (p[n - 1] <> 47) THEN
        _folder := CONCAT(_folder, '\');
    END_IF
END_IF
_where := Where;
_foldersMade := FALSE;
_mkPos := 0;
Setup := TRUE;
END_METHOD

METHOD M_Kind : E_ConfigStore
M_Kind := E_ConfigStore.FILE_JSON;
END_METHOD

METHOD M_Confidential : BOOL
M_Confidential := TRUE;
END_METHOD

METHOD PROTECTED _M_Step : BOOL
VAR
    i : INT;
    best : INT;
    confirmed : UDINT;
    keyPath : STRING(255);
END_VAR
_M_Step := FALSE;
CASE _phase OF
    0:      // a new request: read both headers first, for a read and a write alike
        IF NOT _foldersMade THEN
            _phase := 1;
            RETURN;
        END_IF
        keyPath := CONCAT(_folder, _qKey[_active]);
        _keyCrc := F_Crc32(pData := ADR(keyPath), Size := INT_TO_UDINT(LEN(keyPath)));
        _invalidSeen := FALSE;
        _ioFailed := FALSE;
        FOR i := 1 TO 2 DO
            _hdrValid[i] := FALSE;
        END_FOR
        _slot := 1;
        _phase := 10;
    1:      // create the folder chain, one level per operation
        i := _M_NextSeparator(StartAt := _mkPos);
        IF i < 0 THEN
            _foldersMade := TRUE;
            _phase := 0;
        ELSE
            _mkPos := i + 1;
            _mkdir(bExecute := FALSE);
            _mkdir(sNetId := '', sPathName := LEFT(_folder, i), ePath := _where,
                bExecute := TRUE, tTimeout := IO_TIMEOUT);
            _phase := 2;
        END_IF
    2:
        _mkdir(bExecute := FALSE);
        IF NOT _mkdir.bBusy THEN
            _phase := 1;            // an existing folder answers with an error: ignored
        END_IF

    10:     // header scan: open the slot
        _open(bExecute := FALSE);
        _open(sNetId := '', sPathName := _M_Path(Slot := _slot),
            nMode := Tc2_System.FOPEN_MODEREAD OR Tc2_System.FOPEN_MODEBINARY,
            ePath := _where, bExecute := TRUE, tTimeout := IO_TIMEOUT);
        _phase := 11;
    11:
        _open(bExecute := FALSE);
        IF NOT _open.bBusy THEN
            IF _open.bError THEN
                IF _open.nErrId <> FILE_NOT_FOUND THEN
                    _M_IoFailed(ErrorId := _open.nErrId);   // there, but not readable
                END_IF
                _phase := 16;
            ELSE
                _handle := _open.hFile;
                _phase := 12;
            END_IF
        END_IF
    12:
        MEMSET(destAddr := ADR(_header), fillByte := 0, n := HEADER_BYTES);
        _read(bExecute := FALSE);
        _read(sNetId := '', hFile := _handle, pReadBuff := ADR(_header),
            cbReadLen := HEADER_BYTES, bExecute := TRUE, tTimeout := IO_TIMEOUT);
        _phase := 13;
    13:
        _read(bExecute := FALSE);
        IF NOT _read.bBusy THEN
            IF _read.bError THEN
                _M_IoFailed(ErrorId := _read.nErrId);
            ELSE
                // A short file or a header that does not verify is damaged content.
                _hdrValid[_slot] := (_read.cbRead = HEADER_BYTES) AND _M_ParseHeader(Slot := _slot);
                IF NOT _hdrValid[_slot] THEN
                    _invalidSeen := TRUE;
                END_IF
            END_IF
            _phase := 14;
        END_IF
    14:
        _close(bExecute := FALSE);
        _close(sNetId := '', hFile := _handle, bExecute := TRUE, tTimeout := IO_TIMEOUT);
        _phase := 15;
    15:
        _close(bExecute := FALSE);
        IF NOT _close.bBusy THEN
            IF _close.bError AND (_close.nErrId <> CLOSE_DONE) THEN
                StorageError := _close.nErrId;
                _phase := 14;                       // never leak an open handle
            ELSE
                _handle := 0;
                _phase := 16;
            END_IF
        END_IF
    16:
        IF _slot = 1 THEN
            _slot := 2;
            _phase := 10;
        ELSIF _ioFailed THEN
            // Storage did not answer: never conclude "empty" from that, and never
            // write over a copy that could not be read.
            _qResult[_active].ErrorId := StorageError;
            _M_Finish();
            _M_Step := TRUE;
        ELSIF _qWrite[_active] THEN
            _phase := 40;
        ELSE
            _attempt := 0;
            _phase := 30;
        END_IF

    30:     // read the newest slot still valid; a rejected slot is no longer valid
        IF _attempt < 2 THEN
            _slot := _M_Newest();
        ELSE
            _slot := 0;
        END_IF
        confirmed := _M_ConfirmedGen();
        IF _slot = 0 THEN
            // Nothing valid. Lost when something existed or was confirmed.
            _qResult[_active].Ok := TRUE;
            _qResult[_active].Lost := _invalidSeen OR (confirmed > 0);
            _M_Finish();
            _M_Step := TRUE;
        ELSIF _hdrLen[_slot] > _qSize[_active] THEN
            _qResult[_active].ErrorId := TOO_LARGE;
            _M_Finish();
            _M_Step := TRUE;
        ELSIF _hdrLen[_slot] = 0 THEN
            // A deletion record: nothing there, by intent.
            _qResult[_active].Ok := TRUE;
            _qResult[_active].Lost := confirmed > _hdrGen[_slot];
            _M_Finish();
            _M_Step := TRUE;
        ELSE
            _phase := 31;
        END_IF
    31:
        _open(bExecute := FALSE);
        _open(sNetId := '', sPathName := _M_Path(Slot := _slot),
            nMode := Tc2_System.FOPEN_MODEREAD OR Tc2_System.FOPEN_MODEBINARY,
            ePath := _where, bExecute := TRUE, tTimeout := IO_TIMEOUT);
        _phase := 32;
    32:
        _open(bExecute := FALSE);
        IF NOT _open.bBusy THEN
            IF _open.bError THEN
                _M_IoFailed(ErrorId := _open.nErrId);
                _qResult[_active].ErrorId := StorageError;
                _M_Finish();
                _M_Step := TRUE;
            ELSE
                _handle := _open.hFile;
                _phase := 33;
            END_IF
        END_IF
    33:
        _read(bExecute := FALSE);
        _read(sNetId := '', hFile := _handle, pReadBuff := ADR(_header),
            cbReadLen := HEADER_BYTES, bExecute := TRUE, tTimeout := IO_TIMEOUT);
        _phase := 34;
    34:
        _read(bExecute := FALSE);
        IF NOT _read.bBusy THEN
            IF _read.bError THEN
                _M_IoFailed(ErrorId := _read.nErrId);
                _ioOk := FALSE;
                _phase := 37;
            ELSE
                // The header must still be the one the scan accepted for THIS slot.
                _M_BuildHeader(pDst := ADR(_expect), Generation := _hdrGen[_slot],
                    Length := _hdrLen[_slot], DataCrc := _hdrCrc[_slot]);
                _ioOk := (_read.cbRead = HEADER_BYTES)
                    AND (MEMCMP(pBuf1 := ADR(_header), pBuf2 := ADR(_expect), n := HEADER_BYTES) = 0);
                IF _ioOk THEN
                    _phase := 35;
                ELSE
                    _phase := 37;
                END_IF
            END_IF
        END_IF
    35:
        _read(bExecute := FALSE);
        _read(sNetId := '', hFile := _handle, pReadBuff := _qData[_active],
            cbReadLen := _hdrLen[_slot], bExecute := TRUE, tTimeout := IO_TIMEOUT);
        _phase := 36;
    36:
        _read(bExecute := FALSE);
        IF NOT _read.bBusy THEN
            IF _read.bError THEN
                _M_IoFailed(ErrorId := _read.nErrId);
                _ioOk := FALSE;
            ELSE
                _ioOk := (_read.cbRead = _hdrLen[_slot]);
            END_IF
            _phase := 37;
        END_IF
    37:
        _close(bExecute := FALSE);
        _close(sNetId := '', hFile := _handle, bExecute := TRUE, tTimeout := IO_TIMEOUT);
        _phase := 38;
    38:
        _close(bExecute := FALSE);
        IF NOT _close.bBusy THEN
            IF _close.bError AND (_close.nErrId <> CLOSE_DONE) THEN
                StorageError := _close.nErrId;
                _phase := 37;
            ELSE
                _handle := 0;
                IF _ioFailed THEN
                    _qResult[_active].ErrorId := StorageError;
                    _M_Finish();
                    _M_Step := TRUE;
                ELSIF _ioOk AND (F_Crc32(pData := _qData[_active], Size := _hdrLen[_slot])
                        = _hdrCrc[_slot]) THEN
                    _qResult[_active].Ok := TRUE;
                    _qResult[_active].Found := TRUE;
                    _qResult[_active].Length := _hdrLen[_slot];
                    _qResult[_active].Lost := _M_ConfirmedGen() > _hdrGen[_slot];
                    StorageError := 0;
                    _M_Finish();
                    _M_Step := TRUE;
                ELSE
                    _M_RejectSlot();            // damaged content: try the other slot
                END_IF
            END_IF
        END_IF

    40:     // write into the slot not holding the newest valid copy
        best := _M_Newest();
        _slot := 1;
        IF best = 1 THEN
            _slot := 2;
        END_IF
        _newGen := _M_ConfirmedGen();
        FOR i := 1 TO 2 DO
            IF _hdrValid[i] THEN
                _newGen := MAX(_newGen, _hdrGen[i]);
            END_IF
        END_FOR
        _newGen := _newGen + 1;
        _M_BuildHeader(pDst := ADR(_header), Generation := _newGen, Length := _qSize[_active],
            DataCrc := F_Crc32(pData := _qData[_active], Size := _qSize[_active]));
        _ioOk := TRUE;
        _phase := 41;
    41:
        _open(bExecute := FALSE);
        _open(sNetId := '', sPathName := _M_Path(Slot := _slot),
            nMode := Tc2_System.FOPEN_MODEWRITE OR Tc2_System.FOPEN_MODEBINARY,
            ePath := _where, bExecute := TRUE, tTimeout := IO_TIMEOUT);
        _phase := 42;
    42:
        _open(bExecute := FALSE);
        IF NOT _open.bBusy THEN
            IF _open.bError THEN
                StorageError := _open.nErrId;
                _qResult[_active].ErrorId := _open.nErrId;
                _M_Finish();
                _M_Step := TRUE;
            ELSE
                _handle := _open.hFile;
                _phase := 43;
            END_IF
        END_IF
    43:
        _write(bExecute := FALSE);
        _write(sNetId := '', hFile := _handle, pWriteBuff := ADR(_header),
            cbWriteLen := HEADER_BYTES, bExecute := TRUE, tTimeout := IO_TIMEOUT);
        _phase := 44;
    44:
        _write(bExecute := FALSE);
        IF NOT _write.bBusy THEN
            _ioOk := NOT _write.bError AND (_write.cbWrite = HEADER_BYTES);
            IF _write.bError THEN
                StorageError := _write.nErrId;
            END_IF
            IF _ioOk AND (_qSize[_active] > 0) THEN
                _phase := 45;
            ELSE
                _phase := 47;
            END_IF
        END_IF
    45:
        _write(bExecute := FALSE);
        _write(sNetId := '', hFile := _handle, pWriteBuff := _qData[_active],
            cbWriteLen := _qSize[_active], bExecute := TRUE, tTimeout := IO_TIMEOUT);
        _phase := 46;
    46:
        _write(bExecute := FALSE);
        IF NOT _write.bBusy THEN
            _ioOk := NOT _write.bError AND (_write.cbWrite = _qSize[_active]);
            IF _write.bError THEN
                StorageError := _write.nErrId;
            END_IF
            _phase := 47;
        END_IF
    47:
        _close(bExecute := FALSE);
        _close(sNetId := '', hFile := _handle, bExecute := TRUE, tTimeout := IO_TIMEOUT);
        _phase := 48;
    48:
        _close(bExecute := FALSE);
        IF NOT _close.bBusy THEN
            IF _close.bError AND (_close.nErrId <> CLOSE_DONE) THEN
                StorageError := _close.nErrId;
                _phase := 47;
            ELSE
                _handle := 0;
                // Durable only if the handle closed cleanly as well.
                IF _ioOk AND NOT _close.bError THEN
                    _M_Confirm();
                    _qResult[_active].Ok := TRUE;
                    StorageError := 0;
                ELSE
                    _qResult[_active].ErrorId := StorageError;
                END_IF
                _M_Finish();
                _M_Step := TRUE;
            END_IF
        END_IF
ELSE
    _qResult[_active].ErrorId := INVALID_REQUEST;   // unknown step: fail the request
    _M_Finish();
    _M_Step := TRUE;
END_CASE
END_METHOD

METHOD PRIVATE _M_Finish
IF NOT _qResult[_active].Ok AND (_qResult[_active].ErrorId = 0) THEN
    _qResult[_active].ErrorId := INVALID_REQUEST;
END_IF
_phase := 0;
END_METHOD

// A slot could not be read at all: the request cannot conclude anything about it.
METHOD PRIVATE _M_IoFailed
VAR_INPUT
    ErrorId : UDINT;
END_VAR
_ioFailed := TRUE;
StorageError := ErrorId;
END_METHOD

// The slot's document did not verify: it is damaged, so it stops being a
// candidate and the newest remaining valid slot is tried.
METHOD PRIVATE _M_RejectSlot
_invalidSeen := TRUE;
_hdrValid[_slot] := FALSE;
_attempt := _attempt + 1;
_phase := 30;
END_METHOD

// The slot with the highest valid header generation, 0 when neither is valid.
METHOD PRIVATE _M_Newest : INT
_M_Newest := 0;
IF _hdrValid[1] THEN
    _M_Newest := 1;
END_IF
IF _hdrValid[2] THEN
    IF _M_Newest = 0 THEN
        _M_Newest := 2;
    ELSIF _hdrGen[2] > _hdrGen[1] THEN
        _M_Newest := 2;
    END_IF
END_IF
END_METHOD

// Record the generation just written for this key (the persistent marker).
METHOD PRIVATE _M_Confirm
VAR
    i : INT;
END_VAR
FOR i := 1 TO PL_Fraktal.MAX_PERSIST_KEYS DO
    IF (_confirmedGen[i] > 0) AND (_confirmedKey[i] = _keyCrc) THEN
        _confirmedGen[i] := _newGen;
        RETURN;
    END_IF
END_FOR
FOR i := 1 TO PL_Fraktal.MAX_PERSIST_KEYS DO
    IF _confirmedGen[i] = 0 THEN
        _confirmedKey[i] := _keyCrc;
        _confirmedGen[i] := _newGen;
        RETURN;
    END_IF
END_FOR
END_METHOD

METHOD PRIVATE _M_ConfirmedGen : UDINT
VAR
    i : INT;
END_VAR
_M_ConfirmedGen := 0;
FOR i := 1 TO PL_Fraktal.MAX_PERSIST_KEYS DO
    IF (_confirmedGen[i] > 0) AND (_confirmedKey[i] = _keyCrc) THEN
        _M_ConfirmedGen := _confirmedGen[i];
        RETURN;
    END_IF
END_FOR
END_METHOD

METHOD PRIVATE _M_Path : STRING(255)
VAR_INPUT
    Slot : INT;
END_VAR
IF Slot = 2 THEN
    _M_Path := CONCAT(CONCAT(_folder, _qKey[_active]), '.b');
ELSE
    _M_Path := CONCAT(CONCAT(_folder, _qKey[_active]), '.a');
END_IF
END_METHOD

// Position of the next '\' or '/' at or after StartAt that ends a folder to create,
// -1 when none is left. A drive root ('C:\') and a leading UNC prefix are skipped.
METHOD PRIVATE _M_NextSeparator : INT
VAR_INPUT
    StartAt : INT;
END_VAR
VAR
    p : POINTER TO BYTE;
    i : INT;
END_VAR
_M_NextSeparator := -1;
p := ADR(_folder);
FOR i := MAX(StartAt, 0) TO 159 DO
    IF p[i] = 0 THEN
        RETURN;
    END_IF
    IF ((p[i] = 92) OR (p[i] = 47)) AND (i > 2) THEN
        _M_NextSeparator := i;
        RETURN;
    END_IF
END_FOR
END_METHOD

METHOD PRIVATE _M_BuildHeader
VAR_INPUT
    pDst       : POINTER TO BYTE;
    Generation : UDINT;
    Length     : UDINT;
    DataCrc    : DWORD;
END_VAR
VAR
    text : STRING(80);
END_VAR
text := HEADER_TEXT;
MEMSET(destAddr := pDst, fillByte := 32, n := HEADER_BYTES);
MEMCPY(destAddr := pDst, srcAddr := ADR(text), n := INT_TO_UDINT(LEN(text)));
pDst[HEADER_BYTES - 1] := 10;
_M_PutHex(pDst := pDst + 16, Value := UDINT_TO_DWORD(Generation));
_M_PutHex(pDst := pDst + 27, Value := UDINT_TO_DWORD(Length));
_M_PutHex(pDst := pDst + 38, Value := _keyCrc);
_M_PutHex(pDst := pDst + 49, Value := DataCrc);
_M_PutHex(pDst := pDst + 60, Value := F_Crc32(pData := pDst, Size := HEADER_CRC_SPAN));
END_METHOD

// A header is valid when re-building it from its own fields gives the same 80
// bytes: that checks the labels, the padding, the header CRC and the key in one
// comparison. Its fields are kept per slot; the payload read rebuilds the
// expected header from them for the slot it is reading.
METHOD PRIVATE _M_ParseHeader : BOOL
VAR_INPUT
    Slot : INT;
END_VAR
VAR
    fileGen : DWORD;
    fileLen : DWORD;
    fileKey : DWORD;
    fileCrc : DWORD;
END_VAR
_M_ParseHeader := FALSE;
IF NOT _M_GetHex(pSrc := ADR(_header) + 16, Value := fileGen) THEN RETURN; END_IF
IF NOT _M_GetHex(pSrc := ADR(_header) + 27, Value := fileLen) THEN RETURN; END_IF
IF NOT _M_GetHex(pSrc := ADR(_header) + 38, Value := fileKey) THEN RETURN; END_IF
IF NOT _M_GetHex(pSrc := ADR(_header) + 49, Value := fileCrc) THEN RETURN; END_IF
IF (fileGen = 0) OR (fileKey <> _keyCrc)
OR (DWORD_TO_UDINT(fileLen) > PL_Fraktal.MAX_PERSIST_DOC_BYTES) THEN
    RETURN;
END_IF
_M_BuildHeader(pDst := ADR(_expect), Generation := DWORD_TO_UDINT(fileGen),
    Length := DWORD_TO_UDINT(fileLen), DataCrc := fileCrc);
IF MEMCMP(pBuf1 := ADR(_header), pBuf2 := ADR(_expect), n := HEADER_BYTES) <> 0 THEN
    RETURN;
END_IF
_hdrGen[Slot] := DWORD_TO_UDINT(fileGen);
_hdrLen[Slot] := DWORD_TO_UDINT(fileLen);
_hdrCrc[Slot] := fileCrc;
_M_ParseHeader := TRUE;
END_METHOD

METHOD PRIVATE _M_PutHex
VAR_INPUT
    pDst  : POINTER TO BYTE;
    Value : DWORD;
END_VAR
VAR
    i : INT;
    nibble : BYTE;
END_VAR
FOR i := 0 TO 7 DO
    nibble := DWORD_TO_BYTE(SHR(Value, INT_TO_UINT((7 - i) * 4)) AND DWORD#16#F);
    IF nibble < 10 THEN
        pDst[i] := BYTE#48 + nibble;    // '0'..'9'
    ELSE
        pDst[i] := BYTE#55 + nibble;    // 'A'..'F'
    END_IF
END_FOR
END_METHOD

// Eight upper-case hexadecimal digits at pSrc, exactly as _M_PutHex writes them.
METHOD PRIVATE _M_GetHex : BOOL
VAR_INPUT
    pSrc : POINTER TO BYTE;
END_VAR
VAR_IN_OUT
    Value : DWORD;
END_VAR
VAR
    i : INT;
    c : BYTE;
    acc : DWORD;
END_VAR
_M_GetHex := FALSE;
acc := 0;
FOR i := 0 TO 7 DO
    c := pSrc[i];
    IF (c >= 48) AND (c <= 57) THEN
        acc := SHL(acc, 4) OR (BYTE_TO_DWORD(c) - DWORD#48);
    ELSIF (c >= 65) AND (c <= 70) THEN
        acc := SHL(acc, 4) OR (BYTE_TO_DWORD(c) - DWORD#55);
    ELSE
        RETURN;
    END_IF
END_FOR
Value := acc;
_M_GetHex := TRUE;
END_METHOD

END_FUNCTION_BLOCK

// ---- Connectivity/FB_PersistMediumBase.TcPOU
// Core §3.8b - what every I_PersistMedium shares, written once: the bounded
// request queue, tickets, first-in-first-out service, polling and the key rules.
// A concrete medium supplies M_Kind, M_Confidential and _M_Step, which works on
// the one ACTIVE request (_qKey/_qData/_qSize/_qWrite[_active]) until it is done.
FUNCTION_BLOCK ABSTRACT FB_PersistMediumBase IMPLEMENTS I_PersistMedium
VAR
    _qState  : ARRAY[1..PL_Fraktal.MAX_PERSIST_QUEUE] OF INT;    // FREE/QUEUED/ACTIVE/DONE
    _qTicket : ARRAY[1..PL_Fraktal.MAX_PERSIST_QUEUE] OF UDINT;
    _qKey    : ARRAY[1..PL_Fraktal.MAX_PERSIST_QUEUE] OF STRING(80);
    {attribute 'OPC.UA.DA' := '0'}
    _qData   : ARRAY[1..PL_Fraktal.MAX_PERSIST_QUEUE] OF PVOID;
    _qSize   : ARRAY[1..PL_Fraktal.MAX_PERSIST_QUEUE] OF UDINT;
    _qWrite  : ARRAY[1..PL_Fraktal.MAX_PERSIST_QUEUE] OF BOOL;
    _qResult : ARRAY[1..PL_Fraktal.MAX_PERSIST_QUEUE] OF ST_PersistResult;
    _lastTicket : UDINT;
    _active     : INT;           // queue entry being worked on (0 = none)
END_VAR
VAR CONSTANT
    FREE   : INT := 0;
    QUEUED : INT := 1;
    ACTIVE : INT := 2;
    DONE   : INT := 3;
    INVALID_REQUEST : UDINT := 16#706;   // ADSERR_DEVICE_INVALIDDATA
END_VAR

// no cyclic body: every caller's M_Poll advances the medium

METHOD ABSTRACT M_Kind : E_ConfigStore
END_METHOD

METHOD ABSTRACT M_Confidential : BOOL
END_METHOD

METHOD M_StartWrite : UDINT
VAR_INPUT
    Key   : STRING(80);
    pData : PVOID;
    Size  : UDINT;
END_VAR
M_StartWrite := 0;
IF (Size > PL_Fraktal.MAX_PERSIST_DOC_BYTES) OR ((Size > 0) AND (pData = 0)) THEN
    RETURN;
END_IF
M_StartWrite := _M_Enqueue(Key := Key, pData := pData, Size := Size, Write := TRUE);
END_METHOD

METHOD M_StartRead : UDINT
VAR_INPUT
    Key   : STRING(80);
    pData : PVOID;
    Size  : UDINT;
END_VAR
M_StartRead := 0;
IF (Size = 0) OR (pData = 0) THEN
    RETURN;
END_IF
M_StartRead := _M_Enqueue(Key := Key, pData := pData, Size := Size, Write := FALSE);
END_METHOD

METHOD M_Poll : BOOL
VAR_INPUT
    Ticket : UDINT;
END_VAR
VAR_IN_OUT
    Result : ST_PersistResult;
END_VAR
VAR
    i    : INT;
    pick : INT;
END_VAR
// Start the oldest queued request when idle, then advance the active one.
IF _active = 0 THEN
    pick := 0;
    FOR i := 1 TO PL_Fraktal.MAX_PERSIST_QUEUE DO
        IF _qState[i] = QUEUED THEN
            IF pick = 0 THEN
                pick := i;
            ELSIF _qTicket[i] < _qTicket[pick] THEN
                pick := i;
            END_IF
        END_IF
    END_FOR
    IF pick > 0 THEN
        _active := pick;
        _qState[pick] := ACTIVE;
        MEMSET(destAddr := ADR(_qResult[pick]), fillByte := 0, n := SIZEOF(ST_PersistResult));
    END_IF
END_IF
IF _active > 0 THEN
    IF _M_Step() THEN
        _qState[_active] := DONE;
        _active := 0;
    END_IF
END_IF
// Report on the caller's own ticket.
M_Poll := TRUE;
FOR i := 1 TO PL_Fraktal.MAX_PERSIST_QUEUE DO
    IF (_qState[i] <> FREE) AND (_qTicket[i] = Ticket) THEN
        IF _qState[i] <> DONE THEN
            M_Poll := FALSE;            // still queued or in progress
            RETURN;
        END_IF
        Result := _qResult[i];
        _qState[i] := FREE;
        _qData[i] := 0;
        RETURN;
    END_IF
END_FOR
MEMSET(destAddr := ADR(Result), fillByte := 0, n := SIZEOF(ST_PersistResult));
Result.ErrorId := INVALID_REQUEST;      // unknown or already collected ticket
END_METHOD

METHOD PRIVATE _M_Enqueue : UDINT
VAR_INPUT
    Key   : STRING(80);
    pData : PVOID;
    Size  : UDINT;
    Write : BOOL;
END_VAR
VAR
    i : INT;
END_VAR
_M_Enqueue := 0;
IF NOT F_ValidPersistKey(Key := Key) THEN
    RETURN;
END_IF
FOR i := 1 TO PL_Fraktal.MAX_PERSIST_QUEUE DO
    IF _qState[i] = FREE THEN
        _lastTicket := _lastTicket + 1;
        IF _lastTicket = 0 THEN
            _lastTicket := 1;               // 0 always means refused
        END_IF
        _qTicket[i] := _lastTicket;
        _qKey[i] := Key;
        _qData[i] := pData;
        _qSize[i] := Size;
        _qWrite[i] := Write;
        _qState[i] := QUEUED;
        _M_Enqueue := _lastTicket;
        RETURN;
    END_IF
END_FOR
END_METHOD

// Advance the active request by at most one medium operation. TRUE = finished,
// with _qResult[_active] filled in.
METHOD PROTECTED ABSTRACT _M_Step : BOOL
END_METHOD

END_FUNCTION_BLOCK

// ---- Platform/F_ValidPersistKey.TcPOU
// Core §3.8b - the one rule for an I_PersistMedium document key: a plain name
// of 1 to 80 letters, digits, '_', '.' and '-'. No separator, so on a file
// medium a key can never leave its folder.
FUNCTION F_ValidPersistKey : BOOL
VAR_INPUT
    Key : STRING(80);
END_VAR
VAR
    p : POINTER TO BYTE;
    i : INT;
    c : BYTE;
END_VAR

F_ValidPersistKey := FALSE;
p := ADR(Key);
IF p[0] = 0 THEN
    RETURN;
END_IF
FOR i := 0 TO 79 DO
    c := p[i];
    IF c = 0 THEN
        EXIT;
    END_IF
    IF NOT (((c >= 48) AND (c <= 57)) OR ((c >= 65) AND (c <= 90))
            OR ((c >= 97) AND (c <= 122)) OR (c = 95) OR (c = 46) OR (c = 45)) THEN
        RETURN;
    END_IF
END_FOR
F_ValidPersistKey := TRUE;

END_FUNCTION

// ---- Platform/F_Crc32.TcPOU
// CRC-32/ISO-HDLC (reflected polynomial 0xEDB88320, initial value and final XOR
// 0xFFFFFFFF) over Size bytes at pData: the one implementation behind every
// Fraktal wire record, so a record written natively and one written by the PLC
// are checked by the same arithmetic. Check value: '123456789' -> 0xCBF43926.
// An empty or absent buffer is 0 and is never read.
FUNCTION F_Crc32 : DWORD
VAR_INPUT
    pData : POINTER TO BYTE;
    Size  : UDINT;
END_VAR
VAR
    value    : DWORD;
    index    : UDINT;
    bitIndex : INT;
END_VAR

F_Crc32 := 0;
IF (pData = 0) OR (Size = 0) THEN
    RETURN;
END_IF
value := DWORD#16#FFFFFFFF;
FOR index := 0 TO Size - 1 DO
    value := value XOR BYTE_TO_DWORD(pData[index]);
    FOR bitIndex := 0 TO 7 DO
        IF (value AND DWORD#1) <> 0 THEN
            value := SHR(value, 1) XOR DWORD#16#EDB88320;
        ELSE
            value := SHR(value, 1);
        END_IF
    END_FOR
END_FOR
F_Crc32 := NOT value;

END_FUNCTION

// ---- Platform/F_Sha256.TcPOU
// Core §7.7(c)/§14 - SHA-256 (FIPS 180-4) over Size bytes at pData, in plain ST so
// it needs no crypto library and runs on every TwinCAT the binding supports. Used to
// keep local PINs as salted hashes; it is not a general cryptographic service.
// FALSE = no data pointer (Digest is then zero).
FUNCTION F_Sha256 : BOOL
VAR_INPUT
    pData : POINTER TO BYTE;
    Size  : UDINT;
END_VAR
VAR_IN_OUT
    Digest : ARRAY[0..31] OF BYTE;
END_VAR
VAR
    h      : ARRAY[0..7] OF DWORD;
    w      : ARRAY[0..63] OF DWORD;
    blk    : ARRAY[0..63] OF BYTE;
    padded : UDINT;
    pos    : UDINT;
    b      : UDINT;
    i      : UDINT;
    bitLen : ULINT;
    a, bb, c, d, e, f, g, hh : DWORD;
    s0, s1, t1, t2 : DWORD;
END_VAR
VAR CONSTANT
    K : ARRAY[0..63] OF DWORD := [
        16#428A2F98, 16#71374491, 16#B5C0FBCF, 16#E9B5DBA5, 16#3956C25B, 16#59F111F1, 16#923F82A4, 16#AB1C5ED5,
        16#D807AA98, 16#12835B01, 16#243185BE, 16#550C7DC3, 16#72BE5D74, 16#80DEB1FE, 16#9BDC06A7, 16#C19BF174,
        16#E49B69C1, 16#EFBE4786, 16#0FC19DC6, 16#240CA1CC, 16#2DE92C6F, 16#4A7484AA, 16#5CB0A9DC, 16#76F988DA,
        16#983E5152, 16#A831C66D, 16#B00327C8, 16#BF597FC7, 16#C6E00BF3, 16#D5A79147, 16#06CA6351, 16#14292967,
        16#27B70A85, 16#2E1B2138, 16#4D2C6DFC, 16#53380D13, 16#650A7354, 16#766A0ABB, 16#81C2C92E, 16#92722C85,
        16#A2BFE8A1, 16#A81A664B, 16#C24B8B70, 16#C76C51A3, 16#D192E819, 16#D6990624, 16#F40E3585, 16#106AA070,
        16#19A4C116, 16#1E376C08, 16#2748774C, 16#34B0BCB5, 16#391C0CB3, 16#4ED8AA4A, 16#5B9CCA4F, 16#682E6FF3,
        16#748F82EE, 16#78A5636F, 16#84C87814, 16#8CC70208, 16#90BEFFFA, 16#A4506CEB, 16#BEF9A3F7, 16#C67178F2];
END_VAR

F_Sha256 := FALSE;
FOR i := 0 TO 31 DO
    Digest[i] := 0;
END_FOR
IF pData = 0 THEN
    RETURN;
END_IF
h[0] := 16#6A09E667; h[1] := 16#BB67AE85; h[2] := 16#3C6EF372; h[3] := 16#A54FF53A;
h[4] := 16#510E527F; h[5] := 16#9B05688C; h[6] := 16#1F83D9AB; h[7] := 16#5BE0CD19;
// The message, one 16#80 byte, zeros, then its length in bits (64-bit big-endian),
// padded to whole 64-byte blocks.
padded := ((Size + 9 + 63) / 64) * 64;
bitLen := UDINT_TO_ULINT(Size) * 8;
b := 0;
WHILE b < padded DO
    FOR i := 0 TO 63 DO
        pos := b + i;
        IF pos < Size THEN
            blk[i] := pData[pos];
        ELSIF pos = Size THEN
            blk[i] := 16#80;
        ELSIF pos >= padded - 8 THEN
            blk[i] := ULINT_TO_BYTE(SHR(bitLen, 8 * (padded - 1 - pos)) AND 16#FF);
        ELSE
            blk[i] := 0;
        END_IF
    END_FOR
    FOR i := 0 TO 15 DO
        w[i] := SHL(BYTE_TO_DWORD(blk[4 * i]), 24) OR SHL(BYTE_TO_DWORD(blk[4 * i + 1]), 16)
             OR SHL(BYTE_TO_DWORD(blk[4 * i + 2]), 8) OR BYTE_TO_DWORD(blk[4 * i + 3]);
    END_FOR
    FOR i := 16 TO 63 DO
        s0 := ROR(w[i - 15], 7) XOR ROR(w[i - 15], 18) XOR SHR(w[i - 15], 3);
        s1 := ROR(w[i - 2], 17) XOR ROR(w[i - 2], 19) XOR SHR(w[i - 2], 10);
        w[i] := w[i - 16] + s0 + w[i - 7] + s1;
    END_FOR
    a := h[0]; bb := h[1]; c := h[2]; d := h[3];
    e := h[4]; f := h[5]; g := h[6]; hh := h[7];
    FOR i := 0 TO 63 DO
        s1 := ROR(e, 6) XOR ROR(e, 11) XOR ROR(e, 25);
        t1 := hh + s1 + ((e AND f) XOR ((NOT e) AND g)) + K[i] + w[i];
        s0 := ROR(a, 2) XOR ROR(a, 13) XOR ROR(a, 22);
        t2 := s0 + ((a AND bb) XOR (a AND c) XOR (bb AND c));
        hh := g; g := f; f := e;
        e := d + t1;
        d := c; c := bb; bb := a;
        a := t1 + t2;
    END_FOR
    h[0] := h[0] + a; h[1] := h[1] + bb; h[2] := h[2] + c; h[3] := h[3] + d;
    h[4] := h[4] + e; h[5] := h[5] + f; h[6] := h[6] + g; h[7] := h[7] + hh;
    b := b + 64;
END_WHILE
FOR i := 0 TO 7 DO
    Digest[4 * i]     := DWORD_TO_BYTE(SHR(h[i], 24));
    Digest[4 * i + 1] := DWORD_TO_BYTE(SHR(h[i], 16));
    Digest[4 * i + 2] := DWORD_TO_BYTE(SHR(h[i], 8));
    Digest[4 * i + 3] := DWORD_TO_BYTE(h[i]);
END_FOR
F_Sha256 := TRUE;

END_FUNCTION

// ---- BaseClasses/FB_EngineeringMode.TcPOU
// Core §7.5.1 — the station's commissioning/engineering gate register.
//
// A gate is any deliberate departure from the production configuration: a
// simulation driver in place of the real one, an unverified electrical mapping
// held off, untested logic fenced out — and the §10.5.1 output-force surface.
// Each is a BUILD constant (§7.5.1), so this register is written once at Setup
// and never changes at runtime: declaring a gate IS activating it, and an
// inactive gate is simply never declared. That is why ST_EngineeringGate has no
// `Active` member and why there is no cyclic call to forget (§1.1 O1) — a
// production image registers nothing and this whole surface is empty.
//
// One instance per station, in the composition root, injected into every root
// Unit with FB_UnitBase.SetEngineeringMode. Each Unit then raises the standing
// §7.5.2 annunciation for every registered gate: LOW, SYSTEM, AUTO_RESET,
// not shelvable, and closable only by a build without the gate.
FUNCTION_BLOCK FB_EngineeringMode
VAR_OUTPUT
    Gates : ARRAY[1..PL_Fraktal.MAX_ENGINEERING_GATES] OF ST_EngineeringGate;
    // 0 = a production image: nothing is gated, so nothing is annunciated and
    // no gated surface is published. This is the value a released machine has.
    Count : INT;
    // §10.5.1 rule 1 — the one gate the framework owns rather than the project.
    ForcingActive : BOOL;
    // §7.5.1 bounded register: a station that declares more gates than the table
    // holds would silently stop annunciating the rest, so say so instead (§5.6).
    Truncated : BOOL;
END_VAR
VAR
    _forcingDeclared : BOOL;
END_VAR

// write-once register; no cyclic body

// §7.5.1 — register one ACTIVE gate; returns its slot (0 = not registered).
// `Active` is the caller's BUILD CONSTANT, taken as an input so a composition
// root reads as one line per gate with no IF around it:
//     Engineering.M_Declare(Name := 'USE_SIMULATION',
//         DescriptionKey := 'std.engineering.simulation', Active := USE_SIMULATION);
// Passing a runtime variable here defeats §7.5.1 and is a conformance defect,
// not a shortcut: a gate the machine can switch on is not auditable.
METHOD M_Declare : INT
VAR_INPUT
    Name : STRING(80);
    DescriptionKey : STRING(160);
    Active : BOOL;
END_VAR
VAR
    i : INT;
END_VAR
M_Declare := 0;
IF NOT Active OR (Name = '') THEN
    RETURN;
END_IF
// Idempotent: a re-declared gate keeps its slot, so the framework's own
// M_DeclareOutputForcing and a project that names the same gate cannot produce
// two standing annunciations for one departure.
FOR i := 1 TO Count DO
    IF Gates[i].Name = Name THEN
        M_Declare := i;
        RETURN;
    END_IF
END_FOR
IF Count >= PL_Fraktal.MAX_ENGINEERING_GATES THEN
    Truncated := TRUE;
    RETURN;
END_IF
Count := Count + 1;
Gates[Count].Name := Name;
Gates[Count].DescriptionKey := DescriptionKey;
M_Declare := Count;
END_METHOD

// §10.5.1 rule 1 — register the framework's own force gate from the build
// constant. Called by FB_UnitBase.SetEngineeringMode, so a project that wires
// the register at all gets this gate declared without remembering a second call
// (§1.1 O1); a project that wires nothing simply cannot force (fail closed).
METHOD M_DeclareOutputForcing : BOOL
VAR
    slot : INT;
END_VAR
IF NOT _forcingDeclared THEN
    _forcingDeclared := TRUE;
    slot := M_Declare(Name := 'OUTPUT_FORCING',
        DescriptionKey := 'std.engineering.outputForcing',
        Active := PL_FraktalEngineering.OUTPUT_FORCING);
    // Only a registered gate arms forcing: a full register must not silently
    // grant the capability while failing to annunciate it (§5.6 fail closed).
    ForcingActive := (slot > 0);
END_IF
M_DeclareOutputForcing := ForcingActive;
END_METHOD

END_FUNCTION_BLOCK

// ---- Connectivity/FB_LocalConfigStore.TcPOU
// Core §3.8b — the SHIPPED DEFAULT parameter-set store: named sets of
// (Scope, WriteKey) records held in the PLC's own retentive memory, so a
// conforming station persists its parametrization with no file system, no
// network and no configuration (E_ConfigStore.LOCAL_RETAIN).
//
// It stores RECORDS, not an image. That is not a stylistic choice: §3.8b says a
// byte image of a station's configuration shall not be used, because it
// reinterprets retained bytes silently when a type changes, carries no
// per-value identity for a file/database/MES to bind to, and cannot reject one
// bad value without rejecting all of them. Every value in here is individually
// addressable by (Scope, WriteKey) and is replayed through the owning module's
// typed handler on load, exactly as a single WRITE_CONFIG would be - so a set
// from a slightly different build fails on the one record that no longer fits
// instead of corrupting the machine wholesale.
//
// This store validates NOTHING and authorizes NOTHING (§5.6, §14). It moves
// records. The root owns CONFIG_SET, and the owning module owns the value.
//
// Memory: MAX_CONFIG_SETS × MAX_SET_RECORDS records of ~340 B live in the
// PERSISTENT area, so raising either constant costs the controller's persistent
// budget linearly. A deployment that needs more sets sizes the PLC persistent
// area to match, or substitutes a FILE_JSON/EXTERNAL store.
FUNCTION_BLOCK FB_LocalConfigStore IMPLEMENTS I_ConfigStore
VAR PERSISTENT
    // §3.8b - versioned exactly like every other retained image. Version 0 means
    // never written, so a first boot initializes silently; any other
    // unrecognized version means a real image was rejected and the whole table
    // is cleared rather than read by field position.
    _schema  : UINT;
    _info    : ARRAY[1..PL_Fraktal.MAX_CONFIG_SETS] OF ST_ConfigSetInfo;
    _records : ARRAY[1..PL_Fraktal.MAX_CONFIG_SETS,
                     1..PL_Fraktal.MAX_SET_RECORDS] OF ST_ConfigRecord;
END_VAR
VAR
    // Open save transaction. A set becomes visible only at M_SaveCommit, so a
    // save interrupted by a power loss or a refused record can never leave a
    // half-written set that a later load would apply (§3.8b all-or-nothing).
    _saveSlot   : INT;              // 0 = no save open
    _saveInfo   : ST_ConfigSetInfo;
    _saveCount  : INT;
    _saveFailed : BOOL;
    _staged : FB_ConfigSnapshot;
    _initialized : BOOL;
END_VAR
VAR CONSTANT
    STORE_SCHEMA : UINT := 1;
END_VAR

// No cyclic behaviour: a store is called, never scanned. Every public method
// runs _M_Init first, so the retained-image check cannot be missed by a
// composition root that never calls the instance.
;

// §3.8b - one-shot retained-image check. Exactly the rule every StationCfg
// follows: version 0 initializes silently because nothing was lost; any other
// unrecognized version means a real image was rejected, so the table is cleared
// rather than interpreted by field position. A rejected SET table is reported
// through M_Count going to zero - the sets are simply not there, which is the
// honest answer and the one a client can act on.
METHOD PRIVATE _M_Init
VAR
    i : INT;
END_VAR
IF _initialized THEN
    RETURN;
END_IF
_initialized := TRUE;
IF _schema = STORE_SCHEMA THEN
    RETURN;
END_IF
FOR i := 1 TO PL_Fraktal.MAX_CONFIG_SETS DO
    _info[i].Used := FALSE;
    _info[i].SetName := '';
    _info[i].RecordCount := 0;
END_FOR
_schema := STORE_SCHEMA;
END_METHOD

// Slot holding the named set, or 0. Exact match: a set name is an identity a
// client chose, not a prefix to guess at.
METHOD PRIVATE _M_Find : INT
VAR_INPUT
    SetName : STRING(80);
END_VAR
VAR
    i : INT;
END_VAR
_M_Find := 0;
IF SetName = '' THEN
    RETURN;
END_IF
FOR i := 1 TO PL_Fraktal.MAX_CONFIG_SETS DO
    IF _info[i].Used AND (_info[i].SetName = SetName) THEN
        _M_Find := i;
        RETURN;
    END_IF
END_FOR
END_METHOD

METHOD M_Kind : E_ConfigStore
M_Kind := E_ConfigStore.LOCAL_RETAIN;
END_METHOD

// Open a save. The target slot is chosen now - reusing the one that already
// holds this name, else a free one - but nothing in it is touched until commit.
METHOD M_SaveBegin : BOOL
VAR_INPUT
    Info : ST_ConfigSetInfo;
END_VAR
VAR
    i : INT;
END_VAR
_M_Init();
M_SaveBegin := FALSE;
_saveSlot := 0;
_saveCount := 0;
_saveFailed := FALSE;
IF Info.SetName = '' THEN
    RETURN;
END_IF
_saveSlot := _M_Find(SetName := Info.SetName);
IF _saveSlot = 0 THEN
    FOR i := 1 TO PL_Fraktal.MAX_CONFIG_SETS DO
        IF NOT _info[i].Used THEN
            _saveSlot := i;
            EXIT;
        END_IF
    END_FOR
END_IF
IF _saveSlot = 0 THEN
    RETURN;                               // full: refuse, never evict somebody's set
END_IF
_saveInfo := Info;
_saveInfo.Used := TRUE;
_saveInfo.RecordCount := 0;
M_SaveBegin := _staged.M_SaveBegin(Info := _saveInfo);
END_METHOD

// Stage one record without changing a published set.
METHOD M_SaveRecord : BOOL
VAR_INPUT
    Record : ST_ConfigRecord;
END_VAR
M_SaveRecord := FALSE;
IF _saveSlot = 0 THEN RETURN; END_IF
M_SaveRecord := _staged.M_SaveRecord(Record := Record);
IF NOT M_SaveRecord THEN _saveFailed := TRUE; END_IF
END_METHOD

// Publish only after the complete volatile transaction succeeds.
METHOD M_SaveCommit : BOOL
VAR
    i : INT;
    record : ST_ConfigRecord;
END_VAR
M_SaveCommit := FALSE;
IF (_saveSlot = 0) OR _saveFailed THEN
    M_SaveAbort();
    RETURN;
END_IF
IF NOT _staged.M_SaveCommit() THEN M_SaveAbort(); RETURN; END_IF
IF NOT _staged.M_ReadInfo(SetName := _saveInfo.SetName, Info := _saveInfo) THEN
    M_SaveAbort(); RETURN;
END_IF
// Single-task commit: no fallible storage calls occur after the first copy.
FOR i := 1 TO _saveInfo.RecordCount DO
    _staged.M_ReadRecord(SetName := _saveInfo.SetName, Index := i, Record := record);
    _records[_saveSlot, i] := record;
END_FOR
_info[_saveSlot] := _saveInfo;
_saveSlot := 0;
_saveCount := 0;
M_SaveCommit := TRUE;
END_METHOD

METHOD M_SaveAbort : BOOL
_staged.M_SaveAbort();
_saveSlot := 0;
_saveCount := 0;
_saveFailed := FALSE;
M_SaveAbort := TRUE;
END_METHOD

METHOD M_ReadInfo : BOOL
VAR_INPUT
    SetName : STRING(80);
END_VAR
VAR_IN_OUT
    Info : ST_ConfigSetInfo;
END_VAR
VAR
    slot : INT;
END_VAR
_M_Init();
M_ReadInfo := FALSE;
slot := _M_Find(SetName := SetName);
IF slot = 0 THEN
    RETURN;
END_IF
Info := _info[slot];
M_ReadInfo := TRUE;
END_METHOD

METHOD M_ReadRecord : BOOL
VAR_INPUT
    SetName : STRING(80);
    Index   : INT;
END_VAR
VAR_IN_OUT
    Record : ST_ConfigRecord;
END_VAR
VAR
    slot : INT;
END_VAR
_M_Init();
M_ReadRecord := FALSE;
slot := _M_Find(SetName := SetName);
IF slot = 0 THEN
    RETURN;
END_IF
// Two statements, not one condition: TwinCAT does not short-circuit, so a
// combined test would index _records with an out-of-range Index anyway.
IF (Index < 1) OR (Index > PL_Fraktal.MAX_SET_RECORDS) THEN
    RETURN;
END_IF
IF Index > _info[slot].RecordCount THEN
    RETURN;
END_IF
Record := _records[slot, Index];
M_ReadRecord := TRUE;
END_METHOD

METHOD M_Count : INT
VAR
    i : INT;
END_VAR
_M_Init();
M_Count := 0;
FOR i := 1 TO PL_Fraktal.MAX_CONFIG_SETS DO
    IF _info[i].Used THEN
        M_Count := M_Count + 1;
    END_IF
END_FOR
END_METHOD

// Free the slot. Clearing Used is the single assignment that makes the set
// unreachable, as setting it is what publishes one in M_SaveCommit; the
// records behind it are left to be overwritten by the next save into the slot.
METHOD M_Delete : BOOL
VAR_INPUT
    SetName : STRING(80);
END_VAR
VAR
    slot : INT;
END_VAR
_M_Init();
M_Delete := FALSE;
slot := _M_Find(SetName := SetName);
IF slot = 0 THEN
    RETURN;
END_IF
IF slot = _saveSlot THEN
    RETURN;                               // a save into this slot is open
END_IF
_info[slot].Used := FALSE;
_info[slot].SetName := '';
_info[slot].RecordCount := 0;
M_Delete := TRUE;
END_METHOD

// Index runs over the OCCUPIED sets in slot order, so a client enumerating
// 1..M_Count sees every set exactly once and no empty slots.
METHOD M_InfoAt : BOOL
VAR_INPUT
    Index : INT;
END_VAR
VAR_IN_OUT
    Info : ST_ConfigSetInfo;
END_VAR
VAR
    i    : INT;
    seen : INT;
END_VAR
_M_Init();
M_InfoAt := FALSE;
IF Index < 1 THEN
    RETURN;
END_IF
seen := 0;
FOR i := 1 TO PL_Fraktal.MAX_CONFIG_SETS DO
    IF _info[i].Used THEN
        seen := seen + 1;
        IF seen = Index THEN
            Info := _info[i];
            M_InfoAt := TRUE;
            RETURN;
        END_IF
    END_IF
END_FOR
END_METHOD

END_FUNCTION_BLOCK

// ---- Connectivity/FB_ConfigSnapshot.TcPOU
// Volatile bounded transaction/snapshot storage. No retained set slot is consumed.
FUNCTION_BLOCK FB_ConfigSnapshot IMPLEMENTS I_ConfigStore
VAR
    _info : ST_ConfigSetInfo;
    _records : ARRAY[1..PL_Fraktal.MAX_SET_RECORDS] OF ST_ConfigRecord;
    _count : INT;
    _open : BOOL;
    _failed : BOOL;
END_VAR

;

METHOD M_Kind : E_ConfigStore
M_Kind := E_ConfigStore.LOCAL_RETAIN;
END_METHOD

METHOD M_SaveBegin : BOOL
VAR_INPUT
    Info : ST_ConfigSetInfo;
END_VAR
_info := Info;
_info.Used := FALSE;
_count := 0;
_failed := Info.SetName = '';
_open := NOT _failed;
M_SaveBegin := _open;
END_METHOD

METHOD M_SaveRecord : BOOL
VAR_INPUT
    Record : ST_ConfigRecord;
END_VAR
VAR
    i : INT;
END_VAR
M_SaveRecord := FALSE;
IF NOT _open OR _failed THEN RETURN; END_IF
IF (Record.WriteKey = '') OR (_count >= PL_Fraktal.MAX_SET_RECORDS) THEN
    _failed := TRUE;
    RETURN;
END_IF
FOR i := 1 TO _count DO
    IF (_records[i].Scope = Record.Scope) AND (_records[i].WriteKey = Record.WriteKey) THEN
        _failed := TRUE;
        RETURN;
    END_IF
END_FOR
_count := _count + 1;
_records[_count] := Record;
M_SaveRecord := TRUE;
END_METHOD

METHOD M_SaveCommit : BOOL
M_SaveCommit := _open AND NOT _failed AND (_count > 0);
_open := FALSE;
_info.RecordCount := _count;
_info.Used := M_SaveCommit;
END_METHOD

METHOD M_SaveAbort : BOOL
_open := FALSE;
_info.Used := FALSE;
M_SaveAbort := TRUE;
END_METHOD

METHOD M_ReadInfo : BOOL
VAR_INPUT
    SetName : STRING(80);
END_VAR
VAR_IN_OUT
    Info : ST_ConfigSetInfo;
END_VAR
M_ReadInfo := _info.Used AND (_info.SetName = SetName);
IF M_ReadInfo THEN Info := _info; END_IF
END_METHOD

METHOD M_ReadRecord : BOOL
VAR_INPUT
    SetName : STRING(80);
    Index : INT;
END_VAR
VAR_IN_OUT
    Record : ST_ConfigRecord;
END_VAR
M_ReadRecord := FALSE;
IF NOT _info.Used OR (_info.SetName <> SetName) THEN RETURN; END_IF
IF (Index < 1) OR (Index > _count) THEN RETURN; END_IF
Record := _records[Index];
M_ReadRecord := TRUE;
END_METHOD

METHOD M_Count : INT
M_Count := BOOL_TO_INT(_info.Used);
END_METHOD

METHOD M_Delete : BOOL
VAR_INPUT
    SetName : STRING(80);
END_VAR
M_Delete := _info.Used AND (_info.SetName = SetName);
IF M_Delete THEN _info.Used := FALSE; END_IF
END_METHOD

METHOD M_InfoAt : BOOL
VAR_INPUT
    Index : INT;
END_VAR
VAR_IN_OUT
    Info : ST_ConfigSetInfo;
END_VAR
M_InfoAt := _info.Used AND (Index = 1);
IF M_InfoAt THEN Info := _info; END_IF
END_METHOD

END_FUNCTION_BLOCK

// ---- Connectivity/FB_ConfigSetDocument.TcPOU
// Core §3.8b - one parameter set as a DOCUMENT on an I_PersistMedium: exactly
// the text FB_ConfigSetJson exports (a header line, then one line per record,
// each ended by LF), rendered from and parsed back into any I_ConfigStore.
// Written once and used by both the medium-backed set store and the root's live
// configuration documents, so a set file and a live file are the same format.
//
// Records, not an image (§3.8b): every value keeps its (Scope, WriteKey)
// identity in the file and is replayed through its owner's typed handler. A
// document is parsed completely, or refused - a store sees a set either whole
// or not at all.
FUNCTION_BLOCK FB_ConfigSetDocument
VAR_OUTPUT
    Busy    : BOOL;     // a medium request is in flight
    Ok      : BOOL;     // last request: written durably / the medium answered
    Found   : BOOL;     // last read: a document came back
    Lost    : BOOL;     // last read: the medium lost a document it had confirmed
    ErrorId : UDINT;    // last medium error (0 = none)
END_VAR
VAR
    {attribute 'OPC.UA.DA' := '0'}
    _medium : I_PersistMedium;
    _ticket : UDINT;
    _result : ST_PersistResult;
    _length : UDINT;
    {attribute 'OPC.UA.DA' := '0'}
    _json   : FB_ConfigSetJson;
    {attribute 'OPC.UA.DA' := '0'}
    _doc    : ARRAY[0..PL_Fraktal.MAX_PERSIST_DOC_BYTES - 1] OF BYTE;
END_VAR
VAR CONSTANT
    LINE_MAX : UDINT := 480;
END_VAR

// no cyclic body: the owner calls M_Poll while Busy

// Render the named set of Store and start writing it under Key. FALSE = busy,
// a line the projection refused to render, a document over
// MAX_PERSIST_DOC_BYTES, or a medium that refused the request.
METHOD M_Write : BOOL
VAR_INPUT
    Medium  : I_PersistMedium;
    Key     : STRING(80);
    Store   : I_ConfigStore;
    SetName : STRING(80);
END_VAR
VAR
    info   : ST_ConfigSetInfo;
    record : ST_ConfigRecord;
    line   : STRING(480);
    i      : INT;
END_VAR
M_Write := FALSE;
IF Busy OR (Medium = 0) OR (Store = 0) THEN
    RETURN;
END_IF
ErrorId := 16#705;                          // not rendered (until _M_Start says otherwise)
IF NOT Store.M_ReadInfo(SetName := SetName, Info := info) THEN
    RETURN;
END_IF
_length := 0;
line := _json.M_Header(Info := info);
IF NOT _M_AppendLine(Line := line) THEN
    RETURN;
END_IF
FOR i := 1 TO info.RecordCount DO
    IF NOT Store.M_ReadRecord(SetName := SetName, Index := i, Record := record) THEN
        RETURN;
    END_IF
    line := _json.M_Record(Record := record);
    IF NOT _M_AppendLine(Line := line) THEN
        RETURN;
    END_IF
END_FOR
M_Write := _M_Start(Medium := Medium, Key := Key, Write := TRUE);
END_METHOD

// Start writing an empty document under Key: the set is gone.
METHOD M_Delete : BOOL
VAR_INPUT
    Medium : I_PersistMedium;
    Key    : STRING(80);
END_VAR
M_Delete := FALSE;
IF Busy OR (Medium = 0) THEN
    RETURN;
END_IF
_length := 0;
M_Delete := _M_Start(Medium := Medium, Key := Key, Write := TRUE);
END_METHOD

// Start reading the document under Key; M_Parse takes it once M_Poll is done.
METHOD M_Read : BOOL
VAR_INPUT
    Medium : I_PersistMedium;
    Key    : STRING(80);
END_VAR
M_Read := FALSE;
IF Busy OR (Medium = 0) THEN
    RETURN;
END_IF
_length := 0;
M_Read := _M_Start(Medium := Medium, Key := Key, Write := FALSE);
END_METHOD

// Advance the request. TRUE once nothing is in flight, with the outputs set.
METHOD M_Poll : BOOL
M_Poll := TRUE;
IF NOT Busy THEN
    RETURN;
END_IF
IF NOT _medium.M_Poll(Ticket := _ticket, Result := _result) THEN
    M_Poll := FALSE;
    RETURN;
END_IF
Busy := FALSE;
_ticket := 0;
Ok := _result.Ok;
Found := _result.Found;
Lost := _result.Lost;
ErrorId := _result.ErrorId;
IF Found THEN
    _length := _result.Length;
ELSE
    _length := 0;
END_IF
END_METHOD

// Parse the document last read into Store as one set, and return its header.
// FALSE = not a whole, well-formed set: a line too long, a header or record that
// does not parse, a record count that disagrees, or a store that refused it.
METHOD M_Parse : BOOL
VAR_INPUT
    Store : I_ConfigStore;
END_VAR
VAR_IN_OUT
    Info : ST_ConfigSetInfo;
END_VAR
VAR
    header  : ST_ConfigSetInfo;
    record  : ST_ConfigRecord;
    line    : STRING(480);
    pLine   : POINTER TO BYTE;
    pos     : UDINT;
    n       : UDINT;
    lines   : INT;
    records : INT;
    opened  : BOOL;
END_VAR
M_Parse := FALSE;
IF Busy OR NOT Found OR (Store = 0) OR (_length = 0) THEN
    RETURN;
END_IF
pLine := ADR(line);
pos := 0;
lines := 0;
records := 0;
opened := FALSE;
WHILE pos < _length DO
    n := 0;
    WHILE (pos < _length) AND (_doc[pos] <> 10) DO
        IF n >= LINE_MAX THEN
            IF opened THEN Store.M_SaveAbort(); END_IF
            RETURN;                         // longer than any line we write
        END_IF
        pLine[n] := _doc[pos];
        n := n + 1;
        pos := pos + 1;
    END_WHILE
    pos := pos + 1;                         // past the LF
    IF n > 0 THEN
        IF pLine[n - 1] = 13 THEN
            n := n - 1;                     // tolerate CRLF
        END_IF
    END_IF
    pLine[n] := 0;
    IF n > 0 THEN
        IF lines = 0 THEN
            IF NOT _json.M_ParseHeader(Line := line, Info := header) THEN
                RETURN;
            END_IF
            header.Used := TRUE;
            IF NOT Store.M_SaveBegin(Info := header) THEN
                RETURN;
            END_IF
            opened := TRUE;
        ELSE
            IF NOT _json.M_ParseRecord(Line := line, Record := record) THEN
                Store.M_SaveAbort();
                RETURN;
            END_IF
            IF NOT Store.M_SaveRecord(Record := record) THEN
                Store.M_SaveAbort();
                RETURN;
            END_IF
            records := records + 1;
        END_IF
        lines := lines + 1;
    END_IF
END_WHILE
IF NOT opened THEN
    RETURN;
END_IF
IF records <> header.RecordCount THEN
    Store.M_SaveAbort();
    RETURN;
END_IF
IF NOT Store.M_SaveCommit() THEN
    RETURN;
END_IF
Info := header;
M_Parse := TRUE;
END_METHOD

METHOD PRIVATE _M_Start : BOOL
VAR_INPUT
    Medium : I_PersistMedium;
    Key    : STRING(80);
    Write  : BOOL;
END_VAR
_M_Start := FALSE;
Ok := FALSE;
Found := FALSE;
Lost := FALSE;
IF Write THEN
    _ticket := Medium.M_StartWrite(Key := Key, pData := ADR(_doc), Size := _length);
ELSE
    _ticket := Medium.M_StartRead(Key := Key, pData := ADR(_doc),
        Size := PL_Fraktal.MAX_PERSIST_DOC_BYTES);
END_IF
IF _ticket = 0 THEN
    ErrorId := 16#706;                      // refused: bad key, size or a full queue
    RETURN;
END_IF
_medium := Medium;
ErrorId := 0;
Busy := TRUE;
_M_Start := TRUE;
END_METHOD

// Append one rendered line and its LF. An empty line is a line the projection
// refused to render, so the document is refused rather than written with a hole.
METHOD PRIVATE _M_AppendLine : BOOL
VAR_IN_OUT
    Line : STRING(480);
END_VAR
VAR
    p : POINTER TO BYTE;
    n : UDINT;
END_VAR
_M_AppendLine := FALSE;
p := ADR(Line);
n := 0;
WHILE (n < LINE_MAX) AND (p[n] <> 0) DO
    n := n + 1;
END_WHILE
IF (n = 0) OR ((_length + n + 1) > PL_Fraktal.MAX_PERSIST_DOC_BYTES) THEN
    RETURN;
END_IF
MEMCPY(destAddr := ADR(_doc) + _length, srcAddr := p, n := n);
_length := _length + n;
_doc[_length] := 10;
_length := _length + 1;
_M_AppendLine := TRUE;
END_METHOD

END_FUNCTION_BLOCK

// ---- Platform/FB_ConfigSetJson.TcPOU
// Core §3.8b — the TEXT projection of a parameter set: one JSON object per
// record, one per header. This is what makes a set MOVABLE - to a file, to a
// version-control system, to an asset manager, to another controller - which is
// the whole point of having named sets rather than just retentive memory.
//
// FORMAT DECISION (JSON, and per RECORD rather than per document):
//
//   * JSON over XML because the consumers are a Flutter HMI, a Dart gateway and
//     ordinary MES tooling, all of which parse it natively; nothing in the set
//     needs attributes, namespaces or mixed content.
//
//   * Per RECORD, because §3.8b's central prohibition is the byte image, and
//     the stated reasons are that it carries no per-value identity to bind to
//     and cannot reject one bad value without rejecting all of them. A
//     line-per-record document keeps both properties in the serialization
//     itself: every line is independently identified by (scope, key) and
//     independently rejectable. A single monolithic JSON document would parse
//     back to the same records, but a PLC-side parser for one would need an
//     unbounded buffer and would fail the whole file on one bad character -
//     which is the byte image again, in a friendlier syntax.
//
//   * A line is emitted or refused, NEVER truncated. A line may be 480
//     characters wide, but the standard string functions (CONCAT, LEN, FIND,
//     MID) are specified to 255 and silently cut there, even into a wider
//     target - measured on the runtime, where a 330-character record rendered
//     as 255 bytes. So nothing here uses them on a line: _M_Put appends byte by
//     byte and REFUSES at the width, _M_Length and _M_Find scan to the
//     terminator, and an over-long line produces an empty string the caller
//     must handle, not a silently shortened value (§5.6).
//
// The projection is pure: no state, no I/O, no allocation. Writing the lines to
// a file, an ADS client or an MES connector is a deployment adapter's job
// (§3.15), not the framework's.
FUNCTION_BLOCK FB_ConfigSetJson
VAR CONSTANT
    // A record line holds a STRING(80) scope, a STRING(160) key, a STRING(80)
    // value with every character escaped, and ~70 characters of fixed syntax.
    LINE_MAX : INT := 480;
END_VAR

// Pure projection: called, never scanned.
;

// JSON string-escaping of one field. Only the two characters JSON REQUIRES
// escaping in a plain string are handled - a backslash and a double quote -
// plus control characters, which are replaced rather than emitted raw because a
// stray control byte in a config value would produce a document no parser
// accepts. Ok is FALSE when the result would not fit, and the caller then
// refuses the whole line instead of shipping half a value.
METHOD PRIVATE _M_Escape : STRING(480)
VAR_INPUT
    Text : STRING(255);
END_VAR
VAR_OUTPUT
    Ok : BOOL;
END_VAR
VAR
    pIn  : POINTER TO BYTE;
    pOut : POINTER TO BYTE;
    buf  : STRING(480);
    i    : INT;
    j    : INT;
    n    : INT;
    ch   : BYTE;
END_VAR
Ok := FALSE;
_M_Escape := '';
buf := '';
pIn := ADR(Text);
pOut := ADR(buf);
n := TO_INT(LEN(Text));
j := 0;
FOR i := 0 TO n - 1 DO
    IF j >= (LINE_MAX - 2) THEN
        RETURN;                            // would not fit: refuse, never trim
    END_IF
    ch := pIn[i];
    IF (ch = 16#5C) OR (ch = 16#22) THEN   // backslash, double quote
        pOut[j] := 16#5C;
        j := j + 1;
        pOut[j] := ch;
        j := j + 1;
    ELSIF ch < 16#20 THEN
        pOut[j] := 16#20;                  // control byte -> space (never raw)
        j := j + 1;
    ELSE
        pOut[j] := ch;
        j := j + 1;
    END_IF
END_FOR
pOut[j] := 0;
_M_Escape := buf;
Ok := TRUE;
END_METHOD

// The length of a zero-terminated line, by scanning - LEN stops seeing a
// string at 255. Bounded by LINE_MAX, so a missing terminator cannot run away.
METHOD PRIVATE _M_Length : INT
VAR_INPUT
    pText : POINTER TO BYTE;
END_VAR
_M_Length := 0;
IF pText = 0 THEN
    RETURN;
END_IF
WHILE (_M_Length < LINE_MAX) AND (pText[_M_Length] <> 0) DO
    _M_Length := _M_Length + 1;
END_WHILE
END_METHOD

// Append the zero-terminated text at pText to Line (Used bytes long). FALSE -
// and Line exactly as it was - when the result would exceed LINE_MAX: the
// append is measured first, so it is whole or not at all.
METHOD PRIVATE _M_Put : BOOL
VAR_INPUT
    pText : POINTER TO BYTE;
END_VAR
VAR_IN_OUT
    Line : STRING(480);
    Used : INT;
END_VAR
VAR
    n    : INT;
    i    : INT;
    pOut : POINTER TO BYTE;
END_VAR
_M_Put := FALSE;
n := _M_Length(pText := pText);
IF (Used < 0) OR ((Used + n) > LINE_MAX) THEN
    RETURN;
END_IF
pOut := ADR(Line);
FOR i := 0 TO n - 1 DO
    pOut[Used + i] := pText[i];
END_FOR
Used := Used + n;
pOut[Used] := 0;
_M_Put := TRUE;
END_METHOD

// _M_Put for a short literal or number (at most 255 characters).
METHOD PRIVATE _M_PutText : BOOL
VAR_INPUT
    Text : STRING(255);
END_VAR
VAR_IN_OUT
    Line : STRING(480);
    Used : INT;
END_VAR
_M_PutText := _M_Put(pText := ADR(Text), Line := Line, Used := Used);
END_METHOD

// Append Tail to Line - the one way a set line longer than a request is put
// back together (IMPORT_CONFIG_SET in pieces). FALSE, with Line untouched, when
// the join would exceed LINE_MAX: refused, never truncated.
METHOD M_Join : BOOL
VAR_INPUT
    Tail : STRING(255);
END_VAR
VAR_IN_OUT
    Line : STRING(480);
END_VAR
VAR
    used : INT;
END_VAR
used := _M_Length(pText := ADR(Line));
M_Join := _M_PutText(Text := Tail, Line := Line, Used := used);
END_METHOD

// Render one set record as a JSON object. Empty result = refused (no key, or
// the escaped line would exceed LINE_MAX); the caller shall treat that as a
// failed export rather than writing an empty line.
//
// The revision travels with the record on purpose. §3.8b lists (Scope, WriteKey,
// ValueType, value) as the minimum; carrying the capability revision too is
// what lets a load REJECT a value whose meaning changed since the set was taken,
// instead of replaying an old number into a field that now means something else.
METHOD M_Record : STRING(480)
VAR_INPUT
    Record : ST_ConfigRecord;
END_VAR
VAR
    scopeText : STRING(480);
    keyText   : STRING(480);
    valueText : STRING(480);
    line      : STRING(480);
    used      : INT;
    ok        : BOOL;
END_VAR
M_Record := '';
IF Record.WriteKey = '' THEN
    RETURN;
END_IF
scopeText := _M_Escape(Text := Record.Scope, Ok => ok);
IF NOT ok THEN
    RETURN;
END_IF
keyText := _M_Escape(Text := Record.WriteKey, Ok => ok);
IF NOT ok THEN
    RETURN;
END_IF
valueText := _M_Escape(Text := Record.ValueText, Ok => ok);
IF NOT ok THEN
    RETURN;
END_IF
// Built byte by byte: every append is whole or refused, so the line is
// emitted complete or not at all (see the header on CONCAT).
line := '';
used := 0;
ok := _M_PutText(Text := '{"scope":"', Line := line, Used := used)
    AND_THEN _M_Put(pText := ADR(scopeText), Line := line, Used := used)
    AND_THEN _M_PutText(Text := '","key":"', Line := line, Used := used)
    AND_THEN _M_Put(pText := ADR(keyText), Line := line, Used := used)
    AND_THEN _M_PutText(Text := '","rev":', Line := line, Used := used)
    AND_THEN _M_PutText(Text := UDINT_TO_STRING(Record.Revision), Line := line, Used := used)
    AND_THEN _M_PutText(Text := ',"kind":', Line := line, Used := used)
    AND_THEN _M_PutText(Text := DINT_TO_STRING(TO_DINT(Record.Kind)), Line := line, Used := used)
    AND_THEN _M_PutText(Text := ',"type":', Line := line, Used := used)
    AND_THEN _M_PutText(Text := DINT_TO_STRING(TO_DINT(Record.ValueType)), Line := line, Used := used)
    AND_THEN _M_PutText(Text := ',"value":"', Line := line, Used := used)
    AND_THEN _M_Put(pText := ADR(valueText), Line := line, Used := used)
    AND_THEN _M_PutText(Text := '"}', Line := line, Used := used);
IF ok THEN
    M_Record := line;
END_IF
END_METHOD

